KUKA KRL program: MyProgram_269().src

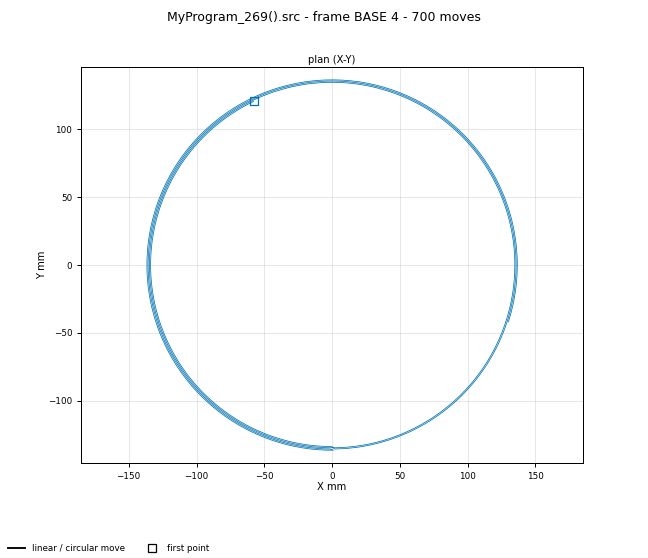
[picture p0: tool path of MyProgram_269().src in frame BASE 4, 700 of 700 moves have a stored position in this frame; points joined in program order, loops and branches not executed]
&ACCESS RVP
&REL 1
&PARAM TEMPLATE = C:\KRC\Roboter\Template\vorgabe
&PARAM EDITMASK = *
DEF MyProgram_269()
; ---- Setting reference (Base) ----
$BASE = BASE_DATA[4]

; --------------------------
; ---- Setting tool (TCP) ----
$TOOL = TOOL_DATA[3]
; --------------------------

$VEL.CP = VEL_APROX_PRINT
Startdeposition()
$VEL.CP = VEL_PRINT
LIN {X -57.9243,Y 120.6655,Z 170,A 116.7349,B 9.9654,C 0.038,E1 9.8949,E2 334.2865} C_DIS
LIN {X -61.6476,Y 118.8079,Z 170,A 118.1625,B 9.9654,C 0.0473,E1 9.8915,E2 332.903} C_DIS
LIN {X -65.3512,Y 116.8125,Z 170,A 119.9699,B 9.9654,C 0.0498,E1 9.887,E2 331.0964} C_DIS
LIN {X -69.0294,Y 114.6773,Z 170,A 121.75,B 9.9654,C 0.0533,E1 9.8828,E2 329.3227} C_DIS
LIN {X -72.8126,Y 112.3129,Z 170,A 123.7286,B 9.9654,C 0.0551,E1 9.8781,E2 327.3377} C_DIS
LIN {X -76.9825,Y 109.497,Z 170,A 126.4571,B 9.9654,C 0.0478,E1 9.8717,E2 324.5421} C_DIS
LIN {X -81.0292,Y 106.5373,Z 170,A 127.9472,B 9.9654,C 0.0641,E1 9.8685,E2 323.1329} C_DIS
LIN {X -83.788,Y 104.3816,Z 170,A 129.5953,B 9.9654,C 0.0641,E1 9.8649,E2 321.4683} C_DIS
LIN {X -86.8669,Y 101.8335,Z 170,A 131.5459,B 9.9654,C 0.0628,E1 9.8607,E2 319.4907} C_DIS
LIN {X -89.382,Y 99.6329,Z 170,A 132.7577,B 9.9653,C 0.0697,E1 9.8582,E2 318.3066} C_DIS
LIN {X -92.6442,Y 96.6073,Z 170,A 134.7532,B 9.9653,C 0.0719,E1 9.8541,E2 316.3021} C_DIS
LIN {X -95.9755,Y 93.2986,Z 170,A 136.5276,B 9.9653,C 0.0805,E1 9.8507,E2 314.5579} C_DIS
LIN {X -98.856,Y 90.2413,Z 170,A 138.5822,B 9.9653,C 0.0797,E1 9.8467,E2 312.4744} C_DIS
LIN {X -101.8694,Y 86.8246,Z 170,A 140.5352,B 9.9652,C 0.084,E1 9.8432,E2 310.5231} C_DIS
LIN {X -104.8688,Y 83.1772,Z 170,A 142.5796,B 9.9652,C 0.0882,E1 9.8396,E2 308.478} C_DIS
LIN {X -107.5965,Y 79.6178,Z 170,A 145.1791,B 9.9652,C 0.0802,E1 9.8351,E2 305.7985} C_DIS
LIN {X -110.8618,Y 75.0035,Z 170,A 147.0989,B 9.9651,C 0.0953,E1 9.8322,E2 303.9418} C_DIS
LIN {X -112.7785,Y 72.0894,Z 170,A 148.8547,B 9.9651,C 0.0943,E1 9.8295,E2 302.156} C_DIS
LIN {X -114.9795,Y 68.5242,Z 170,A 150.0203,B 9.9649,C 0.1102,E1 9.828,E2 301.0679} C_DIS
LIN {X -118.072,Y 63.0474,Z 170,A 152.9817,B 9.9649,C 0.1123,E1 9.8239,E2 298.0773} C_DIS
LIN {X -119.8941,Y 59.5049,Z 170,A 154.6712,B 9.9649,C 0.1171,E1 9.8218,E2 296.3914} C_DIS
LIN {X -121.2827,Y 56.6222,Z 170,A 155.8964,B 9.9648,C 0.1233,E1 9.8203,E2 295.1851} C_DIS
LIN {X -122.7024,Y 53.4752,Z 170,A 157.5597,B 9.9648,C 0.124,E1 9.8184,E2 293.5012} C_DIS
LIN {X -124.0518,Y 50.2648,Z 170,A 158.8105,B 9.9647,C 0.1323,E1 9.8171,E2 292.2806} C_DIS
LIN {X -126.0656,Y 44.9779,Z 170,A 161.6161,B 9.9647,C 0.1321,E1 9.8143,E2 289.4317} C_DIS
LIN {X -127.431,Y 40.9483,Z 170,A 163.3638,B 9.9646,C 0.1385,E1 9.8128,E2 287.6948} C_DIS
LIN {X -128.3886,Y 37.8391,Z 170,A 164.7682,B 9.9646,C 0.1422,E1 9.8117,E2 286.2904} C_DIS
LIN {X -129.2836,Y 34.6579,Z 170,A 166.1835,B 9.9645,C 0.1462,E1 9.8106,E2 284.8766} C_DIS
LIN {X -130.142,Y 31.2805,Z 170,A 167.7247,B 9.9645,C 0.1496,E1 9.8096,E2 283.331} C_DIS
LIN {X -130.9743,Y 27.5965,Z 170,A 169.4193,B 9.9644,C 0.1529,E1 9.8086,E2 281.6288} C_DIS
LIN {X -131.9035,Y 22.7377,Z 170,A 171.5205,B 9.9643,C 0.1592,E1 9.8075,E2 279.5318} C_DIS
LIN {X -132.4714,Y 19.1521,Z 170,A 173.0589,B 9.9642,C 0.164,E1 9.8069,E2 277.9969} C_DIS
LIN {X -132.9158,Y 15.7745,Z 170,A 174.5853,B 9.9642,C 0.167,E1 9.8063,E2 276.4638} C_DIS
LIN {X -133.3417,Y 11.6436,Z 170,A 176.4673,B 9.9641,C 0.1704,E1 9.8058,E2 274.571} C_DIS
LIN {X -133.6571,Y 7.1739,Z 170,A 178.3696,B 9.964,C 0.1762,E1 9.8055,E2 272.6725} C_DIS
LIN {X -133.8021,Y 3.5352,Z 170,A 179.8999,B 9.964,C 0.1813,E1 9.8054,E2 271.1472} C_DIS
LIN {X -133.8485,Y -0.5666,Z 170,A -178.302,B 9.9638,C 0.1857,E1 9.8054,E2 269.3458} C_DIS
LIN {X -133.7769,Y -4.4422,Z 170,A -176.5597,B 9.9638,C 0.189,E1 9.8054,E2 267.595} C_DIS
LIN {X -133.5969,Y -8.205,Z 170,A -174.9767,B 9.9637,C 0.1942,E1 9.8057,E2 266.0171} C_DIS
LIN {X -133.2712,Y -12.4241,Z 170,A -173.1406,B 9.9636,C 0.199,E1 9.8061,E2 264.1797} C_DIS
LIN {X -132.8708,Y -16.1517,Z 170,A -171.4417,B 9.9636,C 0.202,E1 9.8067,E2 262.4708} C_DIS
LIN {X -132.2959,Y -20.3285,Z 170,A -169.3217,B 9.9636,C 0.2015,E1 9.8076,E2 260.3141} C_DIS
LIN {X -131.6934,Y -23.9234,Z 170,A -167.6572,B 9.9635,C 0.2041,E1 9.8084,E2 258.6382} C_DIS
LIN {X -130.9067,Y -27.9095,Z 170,A -166.3798,B 9.9632,C 0.2174,E1 9.8091,E2 257.4187} C_DIS
LIN {X -130.1238,Y -31.3558,Z 170,A -164.4717,B 9.9632,C 0.2145,E1 9.8104,E2 255.4636} C_DIS
LIN {X -129.2659,Y -34.7243,Z 170,A -163.2928,B 9.963,C 0.2242,E1 9.8112,E2 254.3237} C_DIS
LIN {X -127.745,Y -39.9654,Z 170,A -160.7737,B 9.963,C 0.2274,E1 9.8132,E2 251.7842} C_DIS
LIN {X -126.5449,Y -43.6097,Z 170,A -159.228,B 9.9628,C 0.2336,E1 9.8146,E2 250.2517} C_DIS
LIN {X -125.4319,Y -46.7145,Z 170,A -157.8118,B 9.9628,C 0.2374,E1 9.816,E2 248.836} C_DIS
LIN {X -124.3255,Y -49.5857,Z 170,A -156.5337,B 9.9626,C 0.2416,E1 9.8173,E2 247.5636} C_DIS
LIN {X -122.9636,Y -52.8711,Z 170,A -154.9947,B 9.9626,C 0.2453,E1 9.8189,E2 246.0237} C_DIS
LIN {X -121.918,Y -55.2427,Z 170,A -153.2243,B 9.9628,C 0.2361,E1 9.8211,E2 244.1731} C_DIS
LIN {X -119.8678,Y -59.5582,Z 170,A -151.6855,B 9.9624,C 0.2507,E1 9.8229,E2 242.6978} C_DIS
LIN {X -116.8183,Y -65.3408,Z 170,A -148.7983,B 9.9623,C 0.2562,E1 9.8267,E2 239.8017} C_DIS
LIN {X -114.4677,Y -69.3759,Z 170,A -146.8451,B 9.9621,C 0.2619,E1 9.8295,E2 237.8553} C_DIS
LIN {X -112.3203,Y -72.8012,Z 170,A -144.7608,B 9.9621,C 0.2595,E1 9.8327,E2 235.7286} C_DIS
LIN {X -110.2672,Y -75.875,Z 170,A -143.4529,B 9.962,C 0.2683,E1 9.8347,E2 234.4552} C_DIS
LIN {X -107.7234,Y -79.4454,Z 170,A -141.5427,B 9.9619,C 0.272,E1 9.8379,E2 232.5419} C_DIS
LIN {X -104.8133,Y -83.2469,Z 170,A -139.4869,B 9.9617,C 0.2765,E1 9.8414,E2 230.4863} C_DIS
LIN {X -102.0403,Y -86.6235,Z 170,A -137.7705,B 9.9615,C 0.2834,E1 9.8444,E2 228.7897} C_DIS
LIN {X -99.508,Y -89.5215,Z 170,A -136.1827,B 9.9615,C 0.2881,E1 9.8473,E2 227.2099} C_DIS
LIN {X -96.878,Y -92.3609,Z 170,A -134.2445,B 9.9615,C 0.2861,E1 9.8511,E2 225.2379} C_DIS
LIN {X -94.3047,Y -94.9867,Z 170,A -132.5769,B 9.9615,C 0.2874,E1 9.8544,E2 223.5593} C_DIS
LIN {X -89.824,Y -99.2347,Z 170,A -130.0022,B 9.9612,C 0.2938,E1 9.8597,E2 220.9939} C_DIS
LIN {X -86.4166,Y -102.2162,Z 170,A -128.1722,B 9.9611,C 0.2994,E1 9.8635,E2 219.1778} C_DIS
LIN {X -82.174,Y -105.6567,Z 170,A -125.6568,B 9.9611,C 0.3,E1 9.869,E2 216.6411} C_DIS
LIN {X -79.5056,Y -107.6793,Z 170,A -123.9319,B 9.9611,C 0.2967,E1 9.873,E2 214.8805} C_DIS
LIN {X -76.5119,Y -109.8262,Z 170,A -122.6715,B 9.9609,C 0.3054,E1 9.8758,E2 213.6595} C_DIS
LIN {X -73.1187,Y -112.1142,Z 170,A -120.9687,B 9.9608,C 0.309,E1 9.8797,E2 211.9631} C_DIS
LIN {X -69.8846,Y -114.1579,Z 170,A -119.2821,B 9.9608,C 0.3104,E1 9.8837,E2 210.2706} C_DIS
LIN {X -66.9072,Y -115.9281,Z 170,A -117.781,B 9.9607,C 0.312,E1 9.8874,E2 208.7674} C_DIS
LIN {X -63.1609,Y -118.011,Z 170,A -116.0638,B 9.9605,C 0.3168,E1 9.8915,E2 207.0649} C_DIS
LIN {X -59.0597,Y -120.1137,Z 170,A -113.9364,B 9.9605,C 0.3161,E1 9.8969,E2 204.9183} C_DIS
LIN {X -55.1389,Y -121.9644,Z 170,A -112.0625,B 9.9605,C 0.3178,E1 9.9016,E2 203.0422} C_DIS
LIN {X -51.8034,Y -123.4172,Z 170,A -110.4969,B 9.9605,C 0.3192,E1 9.9057,E2 201.4755} C_DIS
LIN {X -49.0158,Y -124.5516,Z 170,A -108.7472,B 9.9607,C 0.311,E1 9.9104,E2 199.6683} C_DIS
LIN {X -44.9288,Y -126.0833,Z 170,A -107.7188,B 9.9601,C 0.3299,E1 9.9128,E2 198.744} C_DIS
LIN {X -38.134,Y -128.3023,Z 170,A -104.2346,B 9.9603,C 0.3236,E1 9.9222,E2 195.2071} C_DIS
LIN {X -34.1836,Y -129.4101,Z 170,A -102.4939,B 9.9603,C 0.325,E1 9.9269,E2 193.468} C_DIS
LIN {X -30.0866,Y -130.4234,Z 170,A -100.6752,B 9.9603,C 0.3258,E1 9.9318,E2 191.6474} C_DIS
LIN {X -26.4187,Y -131.2156,Z 170,A -99.0363,B 9.9603,C 0.3258,E1 9.9363,E2 190.004} C_DIS
LIN {X -22.1834,Y -131.9975,Z 170,A -97.2401,B 9.9603,C 0.3276,E1 9.9412,E2 188.2132} C_DIS
LIN {X -18.358,Y -132.5849,Z 170,A -95.4984,B 9.9603,C 0.3263,E1 9.9461,E2 186.4604} C_DIS
LIN {X -14.1661,Y -133.0969,Z 170,A -93.7824,B 9.9602,C 0.3286,E1 9.9508,E2 184.7551} C_DIS
LIN {X -9.9819,Y -133.4761,Z 170,A -92.0352,B 9.9602,C 0.3299,E1 9.9557,E2 183.0137} C_DIS
LIN {X -5.8315,Y -133.723,Z 170,A -89.4693,B 9.9607,C 0.313,E1 9.9631,E2 180.3486} C_DIS
LIN {X -0.1381,Y -133.85,Z 170,A -87.6713,B 9.9602,C 0.3266,E1 9.9679,E2 178.6297} C_DIS
LIN {X -0.1381,Y -133.85,Z 170,A -87.6713,B 9.9602,C 0.3266,E1 9.9679,E2 178.6297} C_DIS
Enddeposition()
LIN {X 0.9771,Y -134.7546,Z 170,A -87.4135,B 9.7192,C 0.3449,E1 9.728,E2 178.5039} C_DIS
Startdeposition()
$VEL.CP = VEL_PRINT
LIN {X -4.4951,Y -134.6861,Z 170,A -90.2098,B 9.7189,C 0.3551,E1 9.72,E2 181.3599} C_DIS
LIN {X -8.9106,Y -134.467,Z 170,A -92.1285,B 9.7189,C 0.3558,E1 9.7146,E2 183.2843} C_DIS
LIN {X -12.8261,Y -134.1486,Z 170,A -93.73,B 9.7189,C 0.3541,E1 9.7102,E2 184.8779} C_DIS
LIN {X -16.5143,Y -133.7458,Z 170,A -95.3898,B 9.7189,C 0.3555,E1 9.7056,E2 186.5485} C_DIS
LIN {X -20.4759,Y -133.1957,Z 170,A -97.0229,B 9.7189,C 0.3536,E1 9.7011,E2 188.1738} C_DIS
LIN {X -24.06,Y -132.5954,Z 170,A -98.6614,B 9.7189,C 0.3549,E1 9.6965,E2 189.8243} C_DIS
LIN {X -28.2967,Y -131.7559,Z 170,A -100.3974,B 9.7189,C 0.352,E1 9.6918,E2 191.5483} C_DIS
LIN {X -31.5958,Y -131.0038,Z 170,A -101.8668,B 9.7189,C 0.3519,E1 9.6878,E2 193.022} C_DIS
LIN {X -35.6382,Y -129.9641,Z 170,A -103.6858,B 9.7189,C 0.3517,E1 9.6829,E2 194.8468} C_DIS
LIN {X -38.8872,Y -129.0287,Z 170,A -105.798,B 9.7185,C 0.3641,E1 9.677,E2 197.0422} C_DIS
LIN {X -44.1155,Y -127.3346,Z 170,A -107.404,B 9.7191,C 0.3477,E1 9.673,E2 198.5587} C_DIS
LIN {X -47.4018,Y -126.1481,Z 170,A -109.1766,B 9.719,C 0.352,E1 9.6683,E2 200.3669} C_DIS
LIN {X -51.7755,Y -124.4169,Z 170,A -110.9075,B 9.7192,C 0.3448,E1 9.6639,E2 202.0649} C_DIS
LIN {X -54.7429,Y -123.1404,Z 170,A -112.3141,B 9.7192,C 0.344,E1 9.6603,E2 203.4756} C_DIS
LIN {X -57.5955,Y -121.833,Z 170,A -113.5226,B 9.7194,C 0.34,E1 9.6572,E2 204.6686} C_DIS
LIN {X -62.2414,Y -119.5259,Z 170,A -115.9406,B 9.7194,C 0.3415,E1 9.6512,E2 207.1128} C_DIS
LIN {X -66.0211,Y -117.4819,Z 170,A -117.7294,B 9.7194,C 0.3384,E1 9.6468,E2 208.8969} C_DIS
LIN {X -69.3149,Y -115.5697,Z 170,A -119.2947,B 9.7196,C 0.3351,E1 9.643,E2 210.4555} C_DIS
LIN {X -72.4733,Y -113.6153,Z 170,A -121.0175,B 9.7196,C 0.3356,E1 9.6389,E2 212.1957} C_DIS
LIN {X -76.11,Y -111.2118,Z 170,A -122.7076,B 9.7198,C 0.3297,E1 9.635,E2 213.8654} C_DIS
LIN {X -81.907,Y -107.0141,Z 170,A -125.7083,B 9.7199,C 0.3239,E1 9.6283,E2 216.8604} C_DIS
LIN {X -86.3855,Y -103.4331,Z 170,A -128.446,B 9.7199,C 0.3253,E1 9.6223,E2 219.6344} C_DIS
LIN {X -89.9009,Y -100.3922,Z 170,A -130.333,B 9.7201,C 0.32,E1 9.6183,E2 221.5099} C_DIS
LIN {X -93.4041,Y -97.1422,Z 170,A -132.2223,B 9.7203,C 0.3135,E1 9.6145,E2 223.3812} C_DIS
LIN {X -95.7296,Y -94.8507,Z 170,A -133.8096,B 9.7203,C 0.3145,E1 9.6113,E2 224.9924} C_DIS
LIN {X -98.151,Y -92.3427,Z 170,A -135.5462,B 9.7203,C 0.3161,E1 9.6079,E2 226.7595} C_DIS
LIN {X -102.1954,Y -87.8457,Z 170,A -137.9522,B 9.7205,C 0.3077,E1 9.6035,E2 229.1443} C_DIS
LIN {X -105.0155,Y -84.4545,Z 170,A -139.8374,B 9.7205,C 0.3037,E1 9.6002,E2 231.0298} C_DIS
LIN {X -107.7253,Y -80.9697,Z 170,A -141.7675,B 9.7207,C 0.3005,E1 9.5969,E2 232.9655} C_DIS
LIN {X -110.2855,Y -77.4465,Z 170,A -143.6834,B 9.7207,C 0.2974,E1 9.5938,E2 234.8883} C_DIS
LIN {X -113.403,Y -72.8049,Z 170,A -146.0574,B 9.721,C 0.2917,E1 9.5901,E2 237.2606} C_DIS
LIN {X -115.8267,Y -68.8837,Z 170,A -148.0148,B 9.721,C 0.2869,E1 9.5873,E2 239.2166} C_DIS
LIN {X -117.92,Y -65.2354,Z 170,A -150.3141,B 9.721,C 0.2915,E1 9.5841,E2 241.5766} C_DIS
LIN {X -120.0516,Y -61.2196,Z 170,A -151.6792,B 9.7214,C 0.2765,E1 9.5824,E2 242.8716} C_DIS
LIN {X -122.7954,Y -55.5141,Z 170,A -154.5067,B 9.7215,C 0.2719,E1 9.579,E2 245.7139} C_DIS
LIN {X -124.2821,Y -52.0984,Z 170,A -155.9847,B 9.7217,C 0.2659,E1 9.5774,E2 247.1778} C_DIS
LIN {X -125.4871,Y -49.1259,Z 170,A -157.4166,B 9.7217,C 0.2634,E1 9.5759,E2 248.6171} C_DIS
LIN {X -126.5852,Y -46.2249,Z 170,A -158.8446,B 9.7217,C 0.2618,E1 9.5745,E2 250.0574} C_DIS
LIN {X -127.7861,Y -42.7907,Z 170,A -160.2742,B 9.722,C 0.2555,E1 9.5733,E2 251.4716} C_DIS
LIN {X -130,Y -35.5095,Z 170,A -164.2806,B 9.7218,C 0.26,E1 9.5701,E2 255.5684} C_DIS
LIN {X -131.2504,Y -30.5605,Z 170,A -165.8723,B 9.7223,C 0.2439,E1 9.5691,E2 257.0887} C_DIS
LIN {X -132.0168,Y -27.0538,Z 170,A -167.3025,B 9.7224,C 0.2379,E1 9.5683,E2 258.5059} C_DIS
LIN {X -133.1512,Y -20.7629,Z 170,A -170.1331,B 9.7225,C 0.2321,E1 9.5669,E2 261.3479} C_DIS
LIN {X -133.6462,Y -17.2942,Z 170,A -171.6623,B 9.7226,C 0.2285,E1 9.5663,E2 262.8805} C_DIS
LIN {X -134.1146,Y -13.1804,Z 170,A -173.4507,B 9.7227,C 0.2239,E1 9.5658,E2 264.6707} C_DIS
LIN {X -134.4217,Y -9.5513,Z 170,A -175.0694,B 9.7228,C 0.2206,E1 9.5654,E2 266.2964} C_DIS
LIN {X -134.6475,Y -5.5229,Z 170,A -176.7595,B 9.7229,C 0.2152,E1 9.5652,E2 267.9819} C_DIS
LIN {X -134.7544,Y -1.4756,Z 170,A -178.5057,B 9.723,C 0.2106,E1 9.5651,E2 269.7295} C_DIS
LIN {X -134.7396,Y 2.379,Z 170,A 179.7909,B 9.7231,C 0.2069,E1 9.5651,E2 271.439} C_DIS
LIN {X -134.6023,Y 6.5307,Z 170,A 178.0437,B 9.7232,C 0.2015,E1 9.5653,E2 273.1822} C_DIS
LIN {X -134.3987,Y 9.8665,Z 170,A 176.5566,B 9.7232,C 0.1985,E1 9.5656,E2 274.6759} C_DIS
LIN {X -134.0277,Y 14.0378,Z 170,A 174.7855,B 9.7234,C 0.1931,E1 9.5661,E2 276.4441} C_DIS
LIN {X -133.626,Y 17.4478,Z 170,A 173.3066,B 9.7234,C 0.1892,E1 9.5666,E2 277.9238} C_DIS
LIN {X -133.0718,Y 21.2758,Z 170,A 171.3681,B 9.7234,C 0.1896,E1 9.5674,E2 279.8959} C_DIS
LIN {X -132.2236,Y 26.0331,Z 170,A 169.4074,B 9.7236,C 0.182,E1 9.5684,E2 281.8433} C_DIS
LIN {X -131.4843,Y 29.5367,Z 170,A 168.0015,B 9.7237,C 0.1757,E1 9.5693,E2 283.2336} C_DIS
LIN {X -130.6161,Y 33.1621,Z 170,A 166.3806,B 9.7237,C 0.1718,E1 9.5704,E2 284.857} C_DIS
LIN {X -129.5444,Y 37.1365,Z 170,A 164.5101,B 9.7238,C 0.1689,E1 9.5718,E2 286.7402} C_DIS
LIN {X -128.4954,Y 40.6125,Z 170,A 163.0045,B 9.7239,C 0.1639,E1 9.573,E2 288.2395} C_DIS
LIN {X -127.4386,Y 43.8154,Z 170,A 161.1752,B 9.7239,C 0.1668,E1 9.5747,E2 290.1145} C_DIS
LIN {X -126.1073,Y 47.5108,Z 170,A 159.8117,B 9.724,C 0.1569,E1 9.576,E2 291.4397} C_DIS
LIN {X -124.4401,Y 51.72,Z 170,A 158.1735,B 9.7242,C 0.1467,E1 9.5777,E2 293.0415} C_DIS
LIN {X -123.2292,Y 54.5443,Z 170,A 156.5305,B 9.7242,C 0.149,E1 9.5795,E2 294.7234} C_DIS
LIN {X -121.6379,Y 58.0039,Z 170,A 155.0064,B 9.7242,C 0.143,E1 9.5813,E2 296.2345} C_DIS
LIN {X -120.0489,Y 61.225,Z 170,A 153.4683,B 9.7243,C 0.1392,E1 9.5832,E2 297.7722} C_DIS
LIN {X -117.0904,Y 66.7129,Z 170,A 150.7299,B 9.7243,C 0.1339,E1 9.5869,E2 300.5184} C_DIS
LIN {X -115.0176,Y 70.2268,Z 170,A 148.9131,B 9.7244,C 0.131,E1 9.5895,E2 302.3432} C_DIS
LIN {X -112.6799,Y 73.9193,Z 170,A 147.1169,B 9.7244,C 0.1253,E1 9.5922,E2 304.13} C_DIS
LIN {X -108.6836,Y 79.6786,Z 170,A 143.9959,B 9.7245,C 0.1206,E1 9.5973,E2 307.2646} C_DIS
LIN {X -106.0447,Y 83.1583,Z 170,A 142.1258,B 9.7245,C 0.1165,E1 9.6005,E2 309.1344} C_DIS
LIN {X -103.1639,Y 86.7063,Z 170,A 140.1101,B 9.7246,C 0.1134,E1 9.6041,E2 311.1568} C_DIS
LIN {X -100.0761,Y 90.2536,Z 170,A 138.0969,B 9.7246,C 0.1092,E1 9.6078,E2 313.1696} C_DIS
LIN {X -96.8003,Y 93.7575,Z 170,A 136.0795,B 9.7247,C 0.1044,E1 9.6117,E2 315.1822} C_DIS
LIN {X -94.1463,Y 96.4227,Z 170,A 134.4473,B 9.7247,C 0.1017,E1 9.6149,E2 316.8168} C_DIS
LIN {X -90.878,Y 99.5095,Z 170,A 132.4755,B 9.7247,C 0.0989,E1 9.6189,E2 318.7938} C_DIS
LIN {X -87.125,Y 102.8107,Z 170,A 130.3875,B 9.7248,C 0.0941,E1 9.6233,E2 320.8754} C_DIS
LIN {X -83.7824,Y 105.5524,Z 170,A 128.7514,B 9.7249,C 0.087,E1 9.6268,E2 322.4857} C_DIS
LIN {X -78.8326,Y 109.2991,Z 170,A 125.9998,B 9.7249,C 0.0844,E1 9.633,E2 325.2482} C_DIS
LIN {X -75.7767,Y 111.4394,Z 170,A 124.2328,B 9.7249,C 0.085,E1 9.6371,E2 327.0353} C_DIS
LIN {X -72.2613,Y 113.7507,Z 170,A 122.4507,B 9.7249,C 0.082,E1 9.6413,E2 328.815} C_DIS
LIN {X -69.1255,Y 115.6826,Z 170,A 120.8478,B 9.7249,C 0.0803,E1 9.6451,E2 330.4209} C_DIS
LIN {X -65.1242,Y 117.9815,Z 170,A 118.9022,B 9.7249,C 0.0771,E1 9.6498,E2 332.3628} C_DIS
LIN {X -60.4576,Y 120.4376,Z 170,A 116.4291,B 9.7249,C 0.0784,E1 9.6561,E2 334.8614} C_DIS
LIN {X -57.4113,Y 121.9211,Z 170,A 115.2085,B 9.725,C 0.0724,E1 9.6591,E2 336.0547} C_DIS
LIN {X -53.931,Y 123.4987,Z 170,A 113.6182,B 9.725,C 0.0698,E1 9.6631,E2 337.6396} C_DIS
LIN {X -50.2829,Y 125.0276,Z 170,A 110.7916,B 9.7249,C 0.0894,E1 9.6708,E2 340.5996} C_DIS
LIN {X -42.9936,Y 127.7185,Z 170,A 108.5673,B 9.7251,C 0.0658,E1 9.6763,E2 342.6946} C_DIS
LIN {X -34.2182,Y 130.3445,Z 170,A 104.6068,B 9.7251,C 0.0638,E1 9.687,E2 346.6603} C_DIS
LIN {X -30.2257,Y 131.3269,Z 170,A 102.9816,B 9.7251,C 0.0601,E1 9.6913,E2 348.2697} C_DIS
LIN {X -26.7634,Y 132.0759,Z 170,A 101.3934,B 9.7251,C 0.0608,E1 9.6957,E2 349.8667} C_DIS
LIN {X -22.4296,Y 132.8808,Z 170,A 99.5235,B 9.7251,C 0.0597,E1 9.7008,E2 351.7349} C_DIS
LIN {X -18.9606,Y 133.4198,Z 170,A 98.0625,B 9.7251,C 0.0584,E1 9.7048,E2 353.1913} C_DIS
LIN {X -14.9666,Y 133.9278,Z 170,A 96.2689,B 9.7251,C 0.0593,E1 9.7098,E2 354.9937} C_DIS
LIN {X -11.5126,Y 134.2678,Z 170,A 94.9181,B 9.7251,C 0.0564,E1 9.7135,E2 356.3288} C_DIS
LIN {X -8.2991,Y 134.5046,Z 170,A 93.497,B 9.7251,C 0.0571,E1 9.7175,E2 357.7553} C_DIS
LIN {X -4.3993,Y 134.6902,Z 170,A 91.7459,B 9.7251,C 0.0587,E1 9.7224,E2 359.5164} C_DIS
LIN {X -0.5579,Y 134.7595,Z 170,A 90.2192,B 9.7251,C 0.0564,E1 9.7267,E2 361.0297} C_DIS
LIN {X 3.0963,Y 134.7265,Z 170,A 88.5578,B 9.7251,C 0.0586,E1 9.7313,E2 362.7032} C_DIS
LIN {X 7.1572,Y 134.5708,Z 170,A 86.802,B 9.7251,C 0.0594,E1 9.7362,E2 364.4616} C_DIS
LIN {X 11.2305,Y 134.2917,Z 170,A 85.1526,B 9.7251,C 0.0579,E1 9.7408,E2 366.1} C_DIS
LIN {X 15.3754,Y 133.8816,Z 170,A 83.3198,B 9.7251,C 0.0597,E1 9.7459,E2 367.9397} C_DIS
LIN {X 19.2035,Y 133.3851,Z 170,A 81.8206,B 9.7251,C 0.0574,E1 9.75,E2 369.4213} C_DIS
LIN {X 22.3521,Y 132.8937,Z 170,A 80.3941,B 9.7251,C 0.0594,E1 9.754,E2 370.8559} C_DIS
LIN {X 26.5055,Y 132.1284,Z 170,A 78.6392,B 9.7251,C 0.0595,E1 9.7588,E2 372.6055} C_DIS
LIN {X 29.9893,Y 131.3809,Z 170,A 77.108,B 9.7251,C 0.0608,E1 9.7629,E2 374.1382} C_DIS
LIN {X 33.612,Y 130.5019,Z 170,A 75.477,B 9.7251,C 0.0628,E1 9.7674,E2 375.7745} C_DIS
LIN {X 41.0357,Y 128.3602,Z 170,A 72.2905,B 9.7251,C 0.0633,E1 9.7759,E2 378.9487} C_DIS
LIN {X 44.6111,Y 127.1627,Z 170,A 70.4353,B 9.7251,C 0.0702,E1 9.7809,E2 380.8338} C_DIS
LIN {X 48.972,Y 125.5469,Z 170,A 68.7154,B 9.7251,C 0.0667,E1 9.7853,E2 382.5228} C_DIS
LIN {X 52.7591,Y 124.0054,Z 170,A 66.8706,B 9.7251,C 0.0708,E1 9.7901,E2 384.3802} C_DIS
LIN {X 56.2147,Y 122.4757,Z 170,A 65.4282,B 9.7251,C 0.0692,E1 9.7937,E2 385.8029} C_DIS
LIN {X 59.2847,Y 121.0194,Z 170,A 63.9188,B 9.7251,C 0.0723,E1 9.7975,E2 387.3201} C_DIS
LIN {X 62.462,Y 119.4101,Z 170,A 62.4453,B 9.7251,C 0.0734,E1 9.8011,E2 388.7887} C_DIS
LIN {X 66.2679,Y 117.3432,Z 170,A 60.6612,B 9.7251,C 0.0747,E1 9.8055,E2 390.5661} C_DIS
LIN {X 68.8541,Y 115.8444,Z 170,A 59.2954,B 9.725,C 0.0786,E1 9.8088,E2 391.9434} C_DIS
LIN {X 72.4733,Y 113.6153,Z 170,A 57.494,B 9.725,C 0.0812,E1 9.8131,E2 393.7443} C_DIS
LIN {X 78.1668,Y 109.7761,Z 170,A 54.5608,B 9.725,C 0.0863,E1 9.8198,E2 396.6797} C_DIS
LIN {X 81.617,Y 107.2359,Z 170,A 52.6745,B 9.7249,C 0.0908,E1 9.8241,E2 398.5741} C_DIS
LIN {X 85.5189,Y 104.1508,Z 170,A 50.6756,B 9.7249,C 0.092,E1 9.8284,E2 400.5596} C_DIS
LIN {X 88.8945,Y 101.2851,Z 170,A 48.7663,B 9.7249,C 0.0962,E1 9.8324,E2 402.4727} C_DIS
LIN {X 92.3929,Y 98.1037,Z 170,A 46.8346,B 9.7248,C 0.0983,E1 9.8364,E2 404.3955} C_DIS
LIN {X 95.6294,Y 94.9515,Z 170,A 44.8522,B 9.7248,C 0.1036,E1 9.8403,E2 406.386} C_DIS
LIN {X 98.9728,Y 91.4619,Z 170,A 42.8564,B 9.7248,C 0.1065,E1 9.8441,E2 408.3755} C_DIS
LIN {X 101.8721,Y 88.2212,Z 170,A 41.0725,B 9.7247,C 0.109,E1 9.8474,E2 410.1523} C_DIS
LIN {X 103.9422,Y 85.772,Z 170,A 39.1696,B 9.7245,C 0.1243,E1 9.8509,E2 412.1207} C_DIS
LIN {X 107.142,Y 81.7397,Z 170,A 37.5657,B 9.7246,C 0.116,E1 9.8535,E2 413.6554} C_DIS
LIN {X 109.6293,Y 78.372,Z 170,A 35.6235,B 9.7246,C 0.1239,E1 9.8567,E2 415.6181} C_DIS
LIN {X 112.7671,Y 73.7868,Z 170,A 33.4779,B 9.7246,C 0.1245,E1 9.86,E2 417.7388} C_DIS
LIN {X 115.0055,Y 70.2465,Z 170,A 31.7538,B 9.7245,C 0.1276,E1 9.8626,E2 419.4571} C_DIS
LIN {X 117.1796,Y 66.556,Z 170,A 29.6398,B 9.7243,C 0.1389,E1 9.8656,E2 421.6076} C_DIS
LIN {X 118.9531,Y 63.3323,Z 170,A 28.3353,B 9.7243,C 0.1369,E1 9.8672,E2 422.8817} C_DIS
LIN {X 120.6368,Y 60.0603,Z 170,A 26.8561,B 9.7243,C 0.1389,E1 9.8691,E2 424.3515} C_DIS
LIN {X 122.203,Y 56.8043,Z 170,A 25.3984,B 9.7243,C 0.1411,E1 9.8708,E2 425.8007} C_DIS
LIN {X 123.6433,Y 53.5966,Z 170,A 23.9427,B 9.7243,C 0.1441,E1 9.8725,E2 427.2526} C_DIS
LIN {X 125.2323,Y 49.7751,Z 170,A 21.6294,B 9.724,C 0.1618,E1 9.8749,E2 429.6344} C_DIS
LIN {X 126.8753,Y 45.4204,Z 170,A 20.2047,B 9.724,C 0.1542,E1 9.8762,E2 430.9934} C_DIS
LIN {X 128.2042,Y 41.5241,Z 170,A 17.8097,B 9.7237,C 0.1741,E1 9.8784,E2 433.4678} C_DIS
LIN {X 129.7748,Y 36.3151,Z 170,A 16.2523,B 9.7239,C 0.1628,E1 9.8795,E2 434.9355} C_DIS
LIN {X 130.6299,Y 33.1077,Z 170,A 14.841,B 9.7239,C 0.1668,E1 9.8805,E2 436.348} C_DIS
LIN {X 131.5367,Y 29.3071,Z 170,A 13.1174,B 9.7238,C 0.173,E1 9.8816,E2 438.0807} C_DIS
LIN {X 132.3205,Y 25.5275,Z 170,A 11.6108,B 9.7238,C 0.1745,E1 9.8824,E2 439.5722} C_DIS
LIN {X 132.93,Y 22.1345,Z 170,A 10.1412,B 9.7237,C 0.1787,E1 9.8831,E2 441.0435} C_DIS
LIN {X 133.5316,Y 18.1688,Z 170,A 8.5033,B 9.7237,C 0.1821,E1 9.8838,E2 442.6748} C_DIS
LIN {X 133.9501,Y 14.7589,Z 170,A 7.0038,B 9.7235,C 0.1872,E1 9.8843,E2 444.1803} C_DIS
LIN {X 134.298,Y 11.1553,Z 170,A 5.4631,B 9.7235,C 0.1917,E1 9.8846,E2 445.7226} C_DIS
LIN {X 134.5748,Y 7.0779,Z 170,A 3.7664,B 9.7233,C 0.1958,E1 9.8849,E2 447.4159} C_DIS
LIN {X 134.7244,Y 3.1698,Z 170,A 2.0941,B 9.7233,C 0.2008,E1 9.8851,E2 449.091} C_DIS
LIN {X 134.761,Y -0.4414,Z 170,A 0.5387,B 9.7231,C 0.2058,E1 9.8851,E2 450.6503} C_DIS
LIN {X 134.6752,Y -4.8135,Z 170,A -1.0247,B 9.7231,C 0.2042,E1 9.885,E2 452.1792} C_DIS
LIN {X 134.5482,Y -7.5925,Z 170,A -2.4378,B 9.723,C 0.2131,E1 9.8848,E2 453.6218} C_DIS
LIN {X 134.2781,Y -11.3915,Z 170,A -3.9793,B 9.723,C 0.216,E1 9.8844,E2 455.1553} C_DIS
LIN {X 133.8576,Y -15.5767,Z 170,A -5.759,B 9.7228,C 0.221,E1 9.8839,E2 456.9358} C_DIS
LIN {X 133.3506,Y -19.4451,Z 170,A -7.4625,B 9.7227,C 0.2269,E1 9.8832,E2 458.6465} C_DIS
LIN {X 132.6563,Y -23.7196,Z 170,A -9.1637,B 9.7227,C 0.2288,E1 9.8825,E2 460.3324} C_DIS
LIN {X 131.9196,Y -27.5316,Z 170,A -10.9147,B 9.7225,C 0.236,E1 9.8815,E2 462.0975} C_DIS
LIN {X 130.9961,Y -31.6279,Z 170,A -13.3368,B 9.7219,C 0.2561,E1 9.8799,E2 464.5991} C_DIS
LIN {X 129.447,Y -37.4691,Z 170,A -15.0104,B 9.7223,C 0.2422,E1 9.8787,E2 466.166} C_DIS
LIN {X 128.4866,Y -40.6399,Z 170,A -16.4344,B 9.7222,C 0.2466,E1 9.8775,E2 467.5934} C_DIS
LIN {X 127.501,Y -43.6354,Z 170,A -17.9913,B 9.722,C 0.2555,E1 9.8761,E2 469.1784} C_DIS
LIN {X 125.7708,Y -48.3961,Z 170,A -19.8937,B 9.722,C 0.2555,E1 9.8742,E2 471.0521} C_DIS
LIN {X 124.4038,Y -51.807,Z 170,A -21.4219,B 9.7219,C 0.2589,E1 9.8726,E2 472.5777} C_DIS
LIN {X 123.2292,Y -54.5443,Z 170,A -23.6416,B 9.7212,C 0.2848,E1 9.87,E2 474.9156} C_DIS
LIN {X 120.3106,Y -60.7109,Z 170,A -25.6096,B 9.7216,C 0.2706,E1 9.8677,E2 476.7727} C_DIS
LIN {X 118.4923,Y -64.1911,Z 170,A -27.9211,B 9.721,C 0.2901,E1 9.8645,E2 479.1648} C_DIS
LIN {X 115.7314,Y -69.0437,Z 170,A -29.5903,B 9.7213,C 0.2797,E1 9.8623,E2 480.7501} C_DIS
LIN {X 113.5225,Y -72.6183,Z 170,A -31.343,B 9.7213,C 0.2834,E1 9.8597,E2 482.5005} C_DIS
LIN {X 111.2686,Y -76.0273,Z 170,A -33.4986,B 9.7208,C 0.2975,E1 9.8562,E2 484.7095} C_DIS
LIN {X 108.7802,Y -79.547,Z 170,A -34.7233,B 9.7211,C 0.2877,E1 9.8543,E2 485.8612} C_DIS
LIN {X 106.0626,Y -83.1355,Z 170,A -36.8154,B 9.7208,C 0.2964,E1 9.8507,E2 487.9775} C_DIS
LIN {X 103.8118,Y -85.9295,Z 170,A -38.5222,B 9.7206,C 0.3042,E1 9.8477,E2 489.7082} C_DIS
LIN {X 101.6533,Y -88.4726,Z 170,A -39.7263,B 9.7206,C 0.3025,E1 9.8455,E2 490.8875} C_DIS
LIN {X 98.556,Y -91.9103,Z 170,A -41.6939,B 9.7205,C 0.3069,E1 9.8418,E2 492.8571} C_DIS
LIN {X 95.2915,Y -95.2915,Z 170,A -43.3853,B 9.7205,C 0.3041,E1 9.8386,E2 494.5125} C_DIS
LIN {X 92.6636,Y -97.8483,Z 170,A -45.1736,B 9.7203,C 0.3127,E1 9.8349,E2 496.3309} C_DIS
LIN {X 89.3643,Y -100.8702,Z 170,A -47.056,B 9.7203,C 0.3161,E1 9.831,E2 498.2127} C_DIS
LIN {X 86.0826,Y -103.685,Z 170,A -48.8581,B 9.7201,C 0.3189,E1 9.8271,E2 500.0122} C_DIS
LIN {X 80.8541,Y -107.8125,Z 170,A -51.7108,B 9.7199,C 0.3247,E1 9.8209,E2 502.8701} C_DIS
LIN {X 75.7964,Y -111.4261,Z 170,A -54.3343,B 9.7198,C 0.3289,E1 9.8149,E2 505.4937} C_DIS
LIN {X 72.0127,Y -113.9077,Z 170,A -56.1984,B 9.7198,C 0.3308,E1 9.8105,E2 507.3522} C_DIS
LIN {X 65.3454,Y -117.8591,Z 170,A -59.3871,B 9.7196,C 0.3336,E1 9.8028,E2 510.5307} C_DIS
LIN {X 61.6811,Y -119.8167,Z 170,A -61.0631,B 9.7196,C 0.3341,E1 9.7987,E2 512.197} C_DIS
LIN {X 58.9593,Y -121.1799,Z 170,A -62.7075,B 9.7193,C 0.3438,E1 9.7945,E2 513.886} C_DIS
LIN {X 53.8854,Y -123.5184,Z 170,A -64.7938,B 9.7193,C 0.3404,E1 9.7892,E2 515.9384} C_DIS
LIN {X 50.4666,Y -124.9535,Z 170,A -66.6925,B 9.7191,C 0.3495,E1 9.7842,E2 517.8782} C_DIS
LIN {X 47.1541,Y -126.2409,Z 170,A -67.9031,B 9.7192,C 0.3446,E1 9.7812,E2 519.0529} C_DIS
LIN {X 43.5044,Y -127.5464,Z 170,A -69.4883,B 9.7192,C 0.345,E1 9.777,E2 520.6316} C_DIS
LIN {X 39.7151,Y -128.7753,Z 170,A -71.1167,B 9.7192,C 0.3453,E1 9.7727,E2 522.2531} C_DIS
LIN {X 36.1,Y -129.835,Z 170,A -72.8885,B 9.719,C 0.3504,E1 9.7679,E2 524.0471} C_DIS
LIN {X 31.7751,Y -130.9606,Z 170,A -74.6639,B 9.719,C 0.3493,E1 9.7631,E2 525.8084} C_DIS
LIN {X 28.5512,Y -131.701,Z 170,A -76.0798,B 9.719,C 0.3506,E1 9.7592,E2 527.2265} C_DIS
LIN {X 24.47,Y -132.522,Z 170,A -77.9132,B 9.719,C 0.3532,E1 9.7542,E2 529.069} C_DIS
LIN {X 20.6072,Y -133.1753,Z 170,A -79.4899,B 9.719,C 0.3522,E1 9.7499,E2 530.6356} C_DIS
LIN {X 16.8127,Y -133.7093,Z 170,A -81.2382,B 9.7188,C 0.3556,E1 9.745,E2 532.3998} C_DIS
LIN {X 12.9135,Y -134.1402,Z 170,A -82.7788,B 9.7189,C 0.3536,E1 9.7407,E2 533.9255} C_DIS
LIN {X 8.8712,Y -134.4694,Z 170,A -85.0901,B 9.7184,C 0.3666,E1 9.7341,E2 536.3102} C_DIS
LIN {X 4.0559,Y -134.6998,Z 170,A -86.5869,B 9.7189,C 0.3554,E1 9.7301,E2 537.7399} C_DIS
LIN {X 0.9771,Y -134.7546,Z 170,A -87.4108,B 9.7192,C 0.3454,E1 9.728,E2 538.5038} C_DIS
Enddeposition()
LIN {X 0.9771,Y -134.7546,Z 170,A -87.4108,B 9.7192,C 0.3454,E1 9.728,E2 538.5038} C_DIS
Startdeposition()
$VEL.CP = VEL_PRINT
LIN {X 1.5938,Y -135.6645,Z 170,A -86.9648,B 9.6522,C 0.3492,E1 9.6623,E2 538.0882} C_DIS
LIN {X 8.6475,Y -135.3967,Z 170,A -84.0297,B 9.6522,C 0.3495,E1 9.6705,E2 535.1576} C_DIS
LIN {X 12.1264,Y -135.131,Z 170,A -82.4742,B 9.6522,C 0.3472,E1 9.6749,E2 533.5909} C_DIS
LIN {X 15.7984,Y -134.7494,Z 170,A -80.879,B 9.6524,C 0.3457,E1 9.6793,E2 531.9903} C_DIS
LIN {X 18.8367,Y -134.3585,Z 170,A -79.7101,B 9.6523,C 0.3477,E1 9.6825,E2 530.8363} C_DIS
LIN {X 21.4312,Y -133.9704,Z 170,A -78.3746,B 9.6525,C 0.3422,E1 9.6863,E2 529.4714} C_DIS
LIN {X 25.1418,Y -133.3225,Z 170,A -76.9844,B 9.6524,C 0.3455,E1 9.69,E2 528.1055} C_DIS
LIN {X 28.3993,Y -132.6665,Z 170,A -75.5194,B 9.6524,C 0.3432,E1 9.694,E2 526.6318} C_DIS
LIN {X 31.6943,Y -131.918,Z 170,A -74.1043,B 9.6524,C 0.3423,E1 9.6979,E2 525.2172} C_DIS
LIN {X 34.7785,Y -131.1387,Z 170,A -72.6925,B 9.6526,C 0.3396,E1 9.7017,E2 523.7958} C_DIS
LIN {X 38.9856,Y -129.9521,Z 170,A -70.9334,B 9.6526,C 0.3399,E1 9.7064,E2 522.0464} C_DIS
LIN {X 41.7717,Y -129.0822,Z 170,A -69.5361,B 9.6527,C 0.3349,E1 9.7102,E2 520.6273} C_DIS
LIN {X 45.3709,Y -127.8624,Z 170,A -68.1567,B 9.6527,C 0.3383,E1 9.7138,E2 519.2753} C_DIS
LIN {X 48.6481,Y -126.651,Z 170,A -66.5648,B 9.6527,C 0.334,E1 9.718,E2 517.6675} C_DIS
LIN {X 52.1635,Y -125.243,Z 170,A -65.0358,B 9.6527,C 0.3336,E1 9.7219,E2 516.1461} C_DIS
LIN {X 55.1155,Y -123.9725,Z 170,A -63.5972,B 9.6529,C 0.33,E1 9.7256,E2 514.696} C_DIS
LIN {X 59.1306,Y -122.1101,Z 170,A -61.8464,B 9.6529,C 0.3302,E1 9.73,E2 512.9587} C_DIS
LIN {X 62.5616,Y -120.3876,Z 170,A -60.3278,B 9.6529,C 0.3302,E1 9.7337,E2 511.4517} C_DIS
LIN {X 64.9881,Y -119.0962,Z 170,A -58.974,B 9.6531,C 0.3241,E1 9.7371,E2 510.0724} C_DIS
LIN {X 67.6578,Y -117.6006,Z 170,A -57.5222,B 9.6533,C 0.3184,E1 9.7407,E2 508.5993} C_DIS
LIN {X 71.9823,Y -115.0044,Z 170,A -55.6117,B 9.6533,C 0.32,E1 9.7452,E2 506.7147} C_DIS
LIN {X 75.6657,Y -112.6153,Z 170,A -53.9927,B 9.6532,C 0.3222,E1 9.7489,E2 505.1238} C_DIS
LIN {X 78.333,Y -110.776,Z 170,A -52.485,B 9.6533,C 0.3166,E1 9.7524,E2 503.5971} C_DIS
LIN {X 81.4942,Y -108.4718,Z 170,A -50.8499,B 9.6534,C 0.314,E1 9.7561,E2 501.9626} C_DIS
LIN {X 84.8952,Y -105.8313,Z 170,A -48.9243,B 9.6536,C 0.3081,E1 9.7603,E2 500.0217} C_DIS
LIN {X 88.3934,Y -102.9271,Z 170,A -47.0872,B 9.6536,C 0.3062,E1 9.7642,E2 498.1932} C_DIS
LIN {X 91.4696,Y -100.2039,Z 170,A -45.379,B 9.6538,C 0.3033,E1 9.7678,E2 496.4866} C_DIS
LIN {X 94.3303,Y -97.5148,Z 170,A -43.6978,B 9.6538,C 0.2993,E1 9.7712,E2 494.8009} C_DIS
LIN {X 97.4218,Y -94.4264,Z 170,A -41.8847,B 9.654,C 0.2961,E1 9.7747,E2 492.9899} C_DIS
LIN {X 100.3598,Y -91.2978,Z 170,A -40.1329,B 9.654,C 0.2935,E1 9.778,E2 491.2439} C_DIS
LIN {X 103.0897,Y -88.2045,Z 170,A -38.2963,B 9.6542,C 0.2873,E1 9.7814,E2 489.3936} C_DIS
LIN {X 106.1478,Y -84.4985,Z 170,A -36.3268,B 9.6543,C 0.284,E1 9.7849,E2 487.4295} C_DIS
LIN {X 108.899,Y -80.922,Z 170,A -34.4709,B 9.6544,C 0.2806,E1 9.788,E2 485.5778} C_DIS
LIN {X 111.6076,Y -77.1444,Z 170,A -32.5411,B 9.6546,C 0.2766,E1 9.7911,E2 483.6502} C_DIS
LIN {X 114.0326,Y -73.5126,Z 170,A -30.7097,B 9.6546,C 0.2723,E1 9.7939,E2 481.8184} C_DIS
LIN {X 116.3693,Y -69.7542,Z 170,A -28.7071,B 9.6549,C 0.2643,E1 9.7968,E2 479.7969} C_DIS
LIN {X 118.8315,Y -65.4714,Z 170,A -26.8066,B 9.6549,C 0.2634,E1 9.7994,E2 477.9177} C_DIS
LIN {X 120.7591,Y -61.8396,Z 170,A -25.2529,B 9.6549,C 0.2631,E1 9.8014,E2 476.3851} C_DIS
LIN {X 122.2864,Y -58.7617,Z 170,A -23.3961,B 9.6553,C 0.2495,E1 9.8037,E2 474.4754} C_DIS
LIN {X 123.8344,Y -55.4242,Z 170,A -22.3554,B 9.6551,C 0.2577,E1 9.8048,E2 473.4979} C_DIS
LIN {X 124.9527,Y -52.8585,Z 170,A -21.0013,B 9.6553,C 0.2503,E1 9.8063,E2 472.1208} C_DIS
LIN {X 126.3761,Y -49.3554,Z 170,A -19.4502,B 9.6553,C 0.247,E1 9.8079,E2 470.5738} C_DIS
LIN {X 127.7437,Y -45.6999,Z 170,A -17.8417,B 9.6554,C 0.2434,E1 9.8095,E2 468.9686} C_DIS
LIN {X 129.1393,Y -41.5932,Z 170,A -16.1765,B 9.6554,C 0.2423,E1 9.8109,E2 467.3224} C_DIS
LIN {X 130.2117,Y -38.1021,Z 170,A -14.5625,B 9.6556,C 0.2362,E1 9.8122,E2 465.6977} C_DIS
LIN {X 131.6248,Y -32.8941,Z 170,A -12.1641,B 9.6558,C 0.2269,E1 9.8139,E2 463.2819} C_DIS
LIN {X 132.5556,Y -28.913,Z 170,A -10.6041,B 9.6558,C 0.226,E1 9.8149,E2 461.7411} C_DIS
LIN {X 133.1848,Y -25.8622,Z 170,A -9.4723,B 9.6558,C 0.2266,E1 9.8155,E2 460.6309} C_DIS
LIN {X 133.7788,Y -22.5873,Z 170,A -7.9146,B 9.656,C 0.2189,E1 9.8163,E2 459.0527} C_DIS
LIN {X 134.3198,Y -19.1074,Z 170,A -6.4161,B 9.6561,C 0.2143,E1 9.8169,E2 457.5512} C_DIS
LIN {X 134.8629,Y -14.7983,Z 170,A -4.6682,B 9.6561,C 0.2111,E1 9.8175,E2 455.8123} C_DIS
LIN {X 135.1439,Y -11.9735,Z 170,A -3.4852,B 9.6563,C 0.2079,E1 9.8178,E2 454.6301} C_DIS
LIN {X 135.3921,Y -8.7216,Z 170,A -2.2846,B 9.6563,C 0.2082,E1 9.818,E2 453.4503} C_DIS
LIN {X 135.5682,Y -5.3124,Z 170,A -0.6082,B 9.6565,C 0.1983,E1 9.8182,E2 451.7431} C_DIS
LIN {X 135.6703,Y -0.8902,Z 170,A 1.0965,B 9.6565,C 0.1968,E1 9.8182,E2 450.057} C_DIS
LIN {X 135.6496,Y 2.4895,Z 170,A 2.6588,B 9.6566,C 0.1894,E1 9.8182,E2 448.4764} C_DIS
LIN {X 135.5335,Y 6.1667,Z 170,A 4.1898,B 9.6567,C 0.1854,E1 9.8181,E2 446.9468} C_DIS
LIN {X 135.2543,Y 10.667,Z 170,A 6.0903,B 9.6568,C 0.18,E1 9.8177,E2 445.0451} C_DIS
LIN {X 134.9171,Y 14.2953,Z 170,A 7.4025,B 9.6568,C 0.181,E1 9.8173,E2 443.7597} C_DIS
LIN {X 134.5917,Y 17.0959,Z 170,A 8.6112,B 9.6568,C 0.1771,E1 9.8169,E2 442.5477} C_DIS
LIN {X 134.2101,Y 19.8752,Z 170,A 9.9505,B 9.657,C 0.17,E1 9.8164,E2 441.1881} C_DIS
LIN {X 133.6083,Y 23.5758,Z 170,A 11.3802,B 9.657,C 0.1691,E1 9.8157,E2 439.7761} C_DIS
LIN {X 132.9683,Y 26.9506,Z 170,A 12.7867,B 9.657,C 0.1661,E1 9.8149,E2 438.3739} C_DIS
LIN {X 132.3604,Y 29.7957,Z 170,A 14.0526,B 9.6571,C 0.1617,E1 9.8142,E2 437.1023} C_DIS
LIN {X 131.5244,Y 33.2896,Z 170,A 15.5191,B 9.6571,C 0.1586,E1 9.8132,E2 435.6409} C_DIS
LIN {X 130.6299,Y 36.6427,Z 170,A 17.2185,B 9.6573,C 0.149,E1 9.8119,E2 433.9111} C_DIS
LIN {X 129.4187,Y 40.7184,Z 170,A 18.8453,B 9.6573,C 0.148,E1 9.8106,E2 432.3041} C_DIS
LIN {X 128.2232,Y 44.3358,Z 170,A 20.2771,B 9.6573,C 0.1478,E1 9.8093,E2 430.8931} C_DIS
LIN {X 127.3283,Y 46.8504,Z 170,A 21.3975,B 9.6574,C 0.1449,E1 9.8083,E2 429.7727} C_DIS
LIN {X 125.9843,Y 50.3481,Z 170,A 22.9766,B 9.6574,C 0.1407,E1 9.8067,E2 428.1928} C_DIS
LIN {X 124.8252,Y 53.1605,Z 170,A 24.3408,B 9.6575,C 0.1355,E1 9.8052,E2 426.8178} C_DIS
LIN {X 123.3106,Y 56.5814,Z 170,A 25.8345,B 9.6575,C 0.1333,E1 9.8035,E2 425.3337} C_DIS
LIN {X 121.7757,Y 59.8124,Z 170,A 27.3985,B 9.6576,C 0.1281,E1 9.8015,E2 423.762} C_DIS
LIN {X 119.4955,Y 64.2509,Z 170,A 29.9069,B 9.6578,C 0.1133,E1 9.7982,E2 421.2025} C_DIS
LIN {X 117.2583,Y 68.2487,Z 170,A 31.1364,B 9.6577,C 0.1251,E1 9.7966,E2 420.0594} C_DIS
LIN {X 115.6913,Y 70.8723,Z 170,A 32.641,B 9.6577,C 0.1169,E1 9.7944,E2 418.5277} C_DIS
LIN {X 113.3122,Y 74.617,Z 170,A 34.4252,B 9.6578,C 0.1144,E1 9.7917,E2 416.7535} C_DIS
LIN {X 111.1518,Y 77.7996,Z 170,A 36.1273,B 9.6578,C 0.1088,E1 9.789,E2 415.0409} C_DIS
LIN {X 108.5062,Y 81.4486,Z 170,A 38.0126,B 9.6579,C 0.1048,E1 9.7859,E2 413.1569} C_DIS
LIN {X 105.2119,Y 85.6613,Z 170,A 40.2092,B 9.6579,C 0.1011,E1 9.782,E2 410.9669} C_DIS
LIN {X 102.3948,Y 89.0096,Z 170,A 42.0672,B 9.658,C 0.0969,E1 9.7787,E2 409.1068} C_DIS
LIN {X 99.4291,Y 92.3105,Z 170,A 43.8556,B 9.658,C 0.0949,E1 9.7753,E2 407.3283} C_DIS
LIN {X 97.2002,Y 94.6553,Z 170,A 45.2799,B 9.658,C 0.0907,E1 9.7725,E2 405.8963} C_DIS
LIN {X 94.0017,Y 97.8323,Z 170,A 47.0995,B 9.658,C 0.0888,E1 9.7689,E2 404.0864} C_DIS
LIN {X 90.9431,Y 100.6817,Z 170,A 48.883,B 9.6581,C 0.085,E1 9.7652,E2 402.3002} C_DIS
LIN {X 87.5573,Y 103.64,Z 170,A 50.779,B 9.6581,C 0.0815,E1 9.7612,E2 400.404} C_DIS
LIN {X 84.3742,Y 106.2467,Z 170,A 52.4636,B 9.6581,C 0.0796,E1 9.7576,E2 398.7254} C_DIS
LIN {X 80.754,Y 109.0241,Z 170,A 54.3992,B 9.6581,C 0.0761,E1 9.7533,E2 396.7883} C_DIS
LIN {X 77.5066,Y 111.3556,Z 170,A 56.1857,B 9.6582,C 0.0711,E1 9.7492,E2 394.9895} C_DIS
LIN {X 73.2406,Y 114.2067,Z 170,A 58.1864,B 9.6582,C 0.0714,E1 9.7445,E2 393.009} C_DIS
LIN {X 70.7741,Y 115.7515,Z 170,A 59.7123,B 9.6582,C 0.063,E1 9.7408,E2 391.4464} C_DIS
LIN {X 67.5704,Y 117.651,Z 170,A 60.9864,B 9.6582,C 0.0674,E1 9.7378,E2 390.209} C_DIS
LIN {X 63.7978,Y 119.7385,Z 170,A 62.8125,B 9.6582,C 0.0648,E1 9.7333,E2 388.3821} C_DIS
LIN {X 60.634,Y 121.3704,Z 170,A 64.1404,B 9.6582,C 0.0667,E1 9.7301,E2 387.0756} C_DIS
LIN {X 57.4999,Y 122.8859,Z 170,A 65.7595,B 9.6582,C 0.0617,E1 9.7259,E2 385.4383} C_DIS
LIN {X 54.0935,Y 124.4218,Z 170,A 67.2536,B 9.6582,C 0.0617,E1 9.7221,E2 383.9545} C_DIS
LIN {X 49.9144,Y 126.1585,Z 170,A 69.1785,B 9.6583,C 0.0594,E1 9.7172,E2 382.0281} C_DIS
LIN {X 46.4412,Y 127.4765,Z 170,A 70.544,B 9.6583,C 0.0622,E1 9.7137,E2 380.6875} C_DIS
LIN {X 43.172,Y 128.6201,Z 170,A 72.1735,B 9.6583,C 0.0573,E1 9.7093,E2 379.0378} C_DIS
LIN {X 40.1782,Y 129.587,Z 170,A 73.6735,B 9.6583,C 0.0525,E1 9.7053,E2 377.5171} C_DIS
LIN {X 35.9773,Y 130.816,Z 170,A 75.4271,B 9.6583,C 0.0531,E1 9.7006,E2 375.7755} C_DIS
LIN {X 31.9256,Y 131.8622,Z 170,A 77.0137,B 9.6583,C 0.0558,E1 9.6963,E2 374.2112} C_DIS
LIN {X 29.2484,Y 132.4832,Z 170,A 78.3302,B 9.6583,C 0.0518,E1 9.6927,E2 372.8761} C_DIS
LIN {X 25.5154,Y 133.2511,Z 170,A 79.8281,B 9.6583,C 0.0532,E1 9.6886,E2 371.3921} C_DIS
LIN {X 22.2458,Y 133.8358,Z 170,A 81.2515,B 9.6583,C 0.0522,E1 9.6847,E2 369.9667} C_DIS
LIN {X 18.075,Y 134.4634,Z 170,A 83.05,B 9.6583,C 0.0511,E1 9.6797,E2 368.1666} C_DIS
LIN {X 14.7833,Y 134.8646,Z 170,A 84.2367,B 9.6583,C 0.0551,E1 9.6765,E2 367.0064} C_DIS
LIN {X 11.562,Y 135.1787,Z 170,A 85.8018,B 9.6583,C 0.0507,E1 9.6721,E2 365.4177} C_DIS
LIN {X 7.6091,Y 135.4606,Z 170,A 87.5102,B 9.6583,C 0.0497,E1 9.6673,E2 363.7058} C_DIS
LIN {X 3.7459,Y 135.6205,Z 170,A 89.082,B 9.6583,C 0.0509,E1 9.663,E2 362.142} C_DIS
LIN {X -0.3234,Y 135.6726,Z 170,A 90.655,B 9.6583,C 0.0539,E1 9.6586,E2 360.5876} C_DIS
LIN {X -3.6683,Y 135.6227,Z 170,A 92.2257,B 9.6583,C 0.0508,E1 9.6542,E2 358.9983} C_DIS
LIN {X -7.4136,Y 135.4708,Z 170,A 93.9553,B 9.6583,C 0.0481,E1 9.6493,E2 357.2517} C_DIS
LIN {X -11.45,Y 135.1881,Z 170,A 95.4514,B 9.6583,C 0.0528,E1 9.6452,E2 355.7823} C_DIS
LIN {X -13.9754,Y 134.9515,Z 170,A 96.4899,B 9.6583,C 0.0538,E1 9.6423,E2 354.7484} C_DIS
LIN {X -17.5331,Y 134.5344,Z 170,A 98.1011,B 9.6583,C 0.0524,E1 9.6378,E2 353.1261} C_DIS
LIN {X -21.1546,Y 134.0132,Z 170,A 99.6851,B 9.6583,C 0.0524,E1 9.6335,E2 351.5383} C_DIS
LIN {X -25.3718,Y 133.2786,Z 170,A 101.4645,B 9.6583,C 0.0539,E1 9.6286,E2 349.7634} C_DIS
LIN {X -28.2078,Y 132.7079,Z 170,A 102.6423,B 9.6583,C 0.0556,E1 9.6254,E2 348.5918} C_DIS
LIN {X -31.5129,Y 131.9617,Z 170,A 104.1316,B 9.6583,C 0.0554,E1 9.6213,E2 347.0964} C_DIS
LIN {X -34.2297,Y 131.285,Z 170,A 105.6625,B 9.6583,C 0.0495,E1 9.6171,E2 345.5239} C_DIS
LIN {X -37.5984,Y 130.3592,Z 170,A 106.9062,B 9.6583,C 0.0552,E1 9.6138,E2 344.3094} C_DIS
LIN {X -41.1474,Y 129.2817,Z 170,A 108.3576,B 9.6583,C 0.0589,E1 9.61,E2 342.8731} C_DIS
LIN {X -44.9527,Y 128.0093,Z 170,A 109.9885,B 9.6583,C 0.0618,E1 9.6057,E2 341.2513} C_DIS
LIN {X -49.534,Y 126.3066,Z 170,A 112.2745,B 9.6583,C 0.0597,E1 9.5997,E2 338.9399} C_DIS
LIN {X -53.4573,Y 124.6969,Z 170,A 113.9939,B 9.6583,C 0.0631,E1 9.5952,E2 337.2306} C_DIS
LIN {X -56.7182,Y 123.2473,Z 170,A 115.3545,B 9.6583,C 0.0678,E1 9.5918,E2 335.889} C_DIS
LIN {X -64.8205,Y 119.1876,Z 170,A 119.0602,B 9.6582,C 0.0753,E1 9.5827,E2 332.2016} C_DIS
LIN {X -68.166,Y 117.3064,Z 170,A 121.0699,B 9.6582,C 0.0704,E1 9.5777,E2 330.1462} C_DIS
LIN {X -71.8552,Y 115.0835,Z 170,A 122.9024,B 9.6582,C 0.0729,E1 9.5733,E2 328.3137} C_DIS
LIN {X -75.6669,Y 112.6145,Z 170,A 124.6938,B 9.6582,C 0.0784,E1 9.5692,E2 326.5395} C_DIS
LIN {X -78.0045,Y 111.0077,Z 170,A 126.0146,B 9.6582,C 0.0782,E1 9.5661,E2 325.2048} C_DIS
LIN {X -80.7397,Y 109.0347,Z 170,A 127.593,B 9.6582,C 0.0778,E1 9.5625,E2 323.609} C_DIS
LIN {X -84.6898,Y 105.9955,Z 170,A 129.5732,B 9.6582,C 0.084,E1 9.5582,E2 321.646} C_DIS
LIN {X -88.1123,Y 103.1681,Z 170,A 132.0545,B 9.6582,C 0.0763,E1 9.5528,E2 319.0923} C_DIS
LIN {X -92.0032,Y 99.7137,Z 170,A 133.8278,B 9.6581,C 0.0886,E1 9.5492,E2 317.3732} C_DIS
LIN {X -95.6726,Y 96.1982,Z 170,A 135.8658,B 9.6581,C 0.095,E1 9.5452,E2 315.3505} C_DIS
LIN {X -97.8741,Y 93.9579,Z 170,A 137.753,B 9.6581,C 0.0875,E1 9.5414,E2 313.3961} C_DIS
LIN {X -101.2915,Y 90.2634,Z 170,A 139.1075,B 9.6579,C 0.1063,E1 9.5391,E2 312.138} C_DIS
LIN {X -103.5381,Y 87.6771,Z 170,A 140.8643,B 9.6579,C 0.1039,E1 9.5358,E2 310.3449} C_DIS
LIN {X -106.4614,Y 84.1039,Z 170,A 142.8032,B 9.6579,C 0.1086,E1 9.5324,E2 308.4094} C_DIS
LIN {X -109.1236,Y 80.6196,Z 170,A 144.4865,B 9.6578,C 0.116,E1 9.5296,E2 306.7486} C_DIS
LIN {X -111.6101,Y 77.1408,Z 170,A 146.4754,B 9.6578,C 0.117,E1 9.5264,E2 304.7393} C_DIS
LIN {X -114.0029,Y 73.5583,Z 170,A 148.2866,B 9.6578,C 0.1217,E1 9.5236,E2 302.931} C_DIS
LIN {X -116.2431,Y 69.964,Z 170,A 150.1139,B 9.6577,C 0.1254,E1 9.5209,E2 301.1009} C_DIS
LIN {X -118.1908,Y 66.6206,Z 170,A 152.0595,B 9.6577,C 0.1241,E1 9.5182,E2 299.1189} C_DIS
LIN {X -119.8221,Y 63.6385,Z 170,A 153.2371,B 9.6576,C 0.1324,E1 9.5167,E2 297.9743} C_DIS
LIN {X -121.4898,Y 60.3921,Z 170,A 154.5927,B 9.6575,C 0.1397,E1 9.515,E2 296.643} C_DIS
LIN {X -122.6742,Y 57.9499,Z 170,A 156.0382,B 9.6575,C 0.1375,E1 9.5132,E2 295.1622} C_DIS
LIN {X -124.3361,Y 54.2917,Z 170,A 157.6691,B 9.6575,C 0.1432,E1 9.5114,E2 293.5411} C_DIS
LIN {X -125.7053,Y 51.0404,Z 170,A 158.9458,B 9.6573,C 0.151,E1 9.5101,E2 292.2921} C_DIS
LIN {X -127.2501,Y 47.0586,Z 170,A 161.2646,B 9.6573,C 0.1468,E1 9.5077,E2 289.9122} C_DIS
LIN {X -128.3306,Y 44.0259,Z 170,A 162.463,B 9.6573,C 0.1535,E1 9.5066,E2 288.7351} C_DIS
LIN {X -129.6656,Y 39.9215,Z 170,A 164.1817,B 9.6572,C 0.1604,E1 9.5052,E2 287.031} C_DIS
LIN {X -130.6233,Y 36.6666,Z 170,A 165.604,B 9.6571,C 0.1646,E1 9.5041,E2 285.6115} C_DIS
LIN {X -131.3545,Y 33.9591,Z 170,A 166.763,B 9.6571,C 0.1684,E1 9.5033,E2 284.4569} C_DIS
LIN {X -132.238,Y 30.3315,Z 170,A 168.5042,B 9.6571,C 0.17,E1 9.5021,E2 282.6972} C_DIS
LIN {X -133.0506,Y 26.5458,Z 170,A 170.2602,B 9.657,C 0.1726,E1 9.5011,E2 280.928} C_DIS
LIN {X -133.694,Y 23.0959,Z 170,A 171.6356,B 9.6568,C 0.1787,E1 9.5005,E2 279.5674} C_DIS
LIN {X -134.2022,Y 19.9308,Z 170,A 173.1325,B 9.6568,C 0.1801,E1 9.4998,E2 278.0542} C_DIS
LIN {X -134.7203,Y 16.0422,Z 170,A 174.5881,B 9.6567,C 0.1884,E1 9.4993,E2 276.6249} C_DIS
LIN {X -135.1779,Y 11.5705,Z 170,A 176.6588,B 9.6567,C 0.1909,E1 9.4988,E2 274.535} C_DIS
LIN {X -135.4744,Y 7.3429,Z 170,A 178.5253,B 9.6565,C 0.1948,E1 9.4985,E2 272.6609} C_DIS
LIN {X -135.6319,Y 3.3351,Z 170,A -179.7719,B 9.6565,C 0.1996,E1 9.4983,E2 270.9585} C_DIS
LIN {X -135.6706,Y -0.8456,Z 170,A -178.0175,B 9.6563,C 0.2049,E1 9.4983,E2 269.2073} C_DIS
LIN {X -135.583,Y -4.9321,Z 170,A -176.2634,B 9.6563,C 0.2095,E1 9.4984,E2 267.4514} C_DIS
LIN {X -135.4049,Y -8.5132,Z 170,A -174.7083,B 9.6562,C 0.2131,E1 9.4987,E2 265.8927} C_DIS
LIN {X -135.0633,Y -12.8397,Z 170,A -172.8082,B 9.6561,C 0.2172,E1 9.4992,E2 263.986} C_DIS
LIN {X -134.5606,Y -17.3336,Z 170,A -170.9484,B 9.6559,C 0.2236,E1 9.4998,E2 262.134} C_DIS
LIN {X -133.9831,Y -21.3494,Z 170,A -169.0669,B 9.6559,C 0.2256,E1 9.5006,E2 260.2333} C_DIS
LIN {X -133.3702,Y -24.8924,Z 170,A -167.5488,B 9.6558,C 0.2299,E1 9.5013,E2 258.7165} C_DIS
LIN {X -132.6035,Y -28.6915,Z 170,A -166.0494,B 9.6556,C 0.237,E1 9.5022,E2 257.2355} C_DIS
LIN {X -131.9205,Y -31.6836,Z 170,A -164.5834,B 9.6556,C 0.2376,E1 9.5031,E2 255.7495} C_DIS
LIN {X -129.8903,Y -39.1873,Z 170,A -161.1146,B 9.6554,C 0.2434,E1 9.5058,E2 252.2604} C_DIS
LIN {X -128.1153,Y -44.6469,Z 170,A -158.8563,B 9.6552,C 0.253,E1 9.5078,E2 250.0246} C_DIS
LIN {X -126.5731,Y -48.8485,Z 170,A -157.0909,B 9.655,C 0.2604,E1 9.5095,E2 248.2761} C_DIS
LIN {X -125.2973,Y -52.0335,Z 170,A -155.5329,B 9.655,C 0.2623,E1 9.5111,E2 246.7056} C_DIS
LIN {X -124.0296,Y -54.9879,Z 170,A -154.3034,B 9.6548,C 0.2681,E1 9.5125,E2 245.493} C_DIS
LIN {X -122.5838,Y -58.1391,Z 170,A -152.6024,B 9.6548,C 0.2677,E1 9.5145,E2 243.7636} C_DIS
LIN {X -120.9802,Y -61.4053,Z 170,A -151.0429,B 9.6548,C 0.2712,E1 9.5165,E2 242.2022} C_DIS
LIN {X -118.7914,Y -65.5439,Z 170,A -149.0046,B 9.6546,C 0.2751,E1 9.5192,E2 240.1576} C_DIS
LIN {X -116.6529,Y -69.2784,Z 170,A -147.1471,B 9.6545,C 0.2788,E1 9.5218,E2 238.2962} C_DIS
LIN {X -113.9722,Y -73.6057,Z 170,A -144.3836,B 9.6547,C 0.2727,E1 9.5261,E2 235.4569} C_DIS
LIN {X -110.9727,Y -78.054,Z 170,A -142.8531,B 9.6541,C 0.2916,E1 9.5284,E2 234.0199} C_DIS
LIN {X -108.2084,Y -81.8432,Z 170,A -140.7067,B 9.6541,C 0.293,E1 9.532,E2 231.8538} C_DIS
LIN {X -105.5774,Y -85.2101,Z 170,A -138.8697,B 9.654,C 0.2964,E1 9.5352,E2 230.0136} C_DIS
LIN {X -102.8702,Y -88.4595,Z 170,A -137.0645,B 9.6539,C 0.2999,E1 9.5384,E2 228.2068} C_DIS
LIN {X -100.1168,Y -91.5647,Z 170,A -135.293,B 9.6538,C 0.3032,E1 9.5417,E2 226.4337} C_DIS
LIN {X -97.167,Y -94.6895,Z 170,A -133.4331,B 9.6537,C 0.306,E1 9.5453,E2 224.5688} C_DIS
LIN {X -93.979,Y -97.854,Z 170,A -131.5073,B 9.6536,C 0.3092,E1 9.5492,E2 222.64} C_DIS
LIN {X -90.6423,Y -100.9522,Z 170,A -129.5769,B 9.6535,C 0.3127,E1 9.5532,E2 220.7093} C_DIS
LIN {X -87.2136,Y -103.9285,Z 170,A -127.544,B 9.6535,C 0.3139,E1 9.5575,E2 218.6624} C_DIS
LIN {X -83.2924,Y -107.097,Z 170,A -125.4941,B 9.6533,C 0.3191,E1 9.562,E2 216.6229} C_DIS
LIN {X -78.8078,Y -110.4386,Z 170,A -123.1431,B 9.6531,C 0.3231,E1 9.5673,E2 214.2737} C_DIS
LIN {X -75.3051,Y -112.8561,Z 170,A -121.3418,B 9.6531,C 0.3258,E1 9.5715,E2 212.4722} C_DIS
LIN {X -71.2611,Y -115.4526,Z 170,A -119.2486,B 9.653,C 0.3275,E1 9.5764,E2 210.3713} C_DIS
LIN {X -67.6101,Y -117.6282,Z 170,A -117.435,B 9.653,C 0.3296,E1 9.5808,E2 208.5555} C_DIS
LIN {X -64.0655,Y -119.5951,Z 170,A -115.8198,B 9.6528,C 0.3337,E1 9.5847,E2 206.9526} C_DIS
LIN {X -61.6758,Y -120.8425,Z 170,A -114.6035,B 9.6528,C 0.3336,E1 9.5878,E2 205.7264} C_DIS
LIN {X -57.6594,Y -122.8122,Z 170,A -112.6874,B 9.6528,C 0.3352,E1 9.5926,E2 203.8069} C_DIS
LIN {X -54.2917,Y -124.3361,Z 170,A -111.2361,B 9.6526,C 0.3391,E1 9.5963,E2 202.3693} C_DIS
LIN {X -51.0106,Y -125.7173,Z 170,A -109.7624,B 9.6526,C 0.3412,E1 9.6001,E2 200.8993} C_DIS
LIN {X -48.4343,Y -126.7341,Z 170,A -108.3947,B 9.6526,C 0.3383,E1 9.6037,E2 199.5066} C_DIS
LIN {X -44.7716,Y -128.0721,Z 170,A -106.9111,B 9.6524,C 0.343,E1 9.6075,E2 198.0433} C_DIS
LIN {X -40.5902,Y -129.4597,Z 170,A -104.853,B 9.6525,C 0.3405,E1 9.6131,E2 195.9601} C_DIS
LIN {X -36.3527,Y -130.711,Z 170,A -103.1273,B 9.6524,C 0.3446,E1 9.6177,E2 194.2517} C_DIS
LIN {X -32.6317,Y -131.6914,Z 170,A -101.4904,B 9.6524,C 0.3454,E1 9.6221,E2 192.613} C_DIS
LIN {X -29.4519,Y -132.4389,Z 170,A -100.018,B 9.6524,C 0.3442,E1 9.6261,E2 191.1285} C_DIS
LIN {X -25.7141,Y -133.2131,Z 170,A -98.504,B 9.6524,C 0.3469,E1 9.6303,E2 189.6264} C_DIS
LIN {X -22.4944,Y -133.7944,Z 170,A -97.2214,B 9.6522,C 0.3495,E1 9.6338,E2 188.3559} C_DIS
LIN {X -19.361,Y -134.2836,Z 170,A -95.8352,B 9.6522,C 0.3489,E1 9.6376,E2 186.9633} C_DIS
LIN {X -16.6923,Y -134.6428,Z 170,A -94.7185,B 9.6522,C 0.3496,E1 9.6407,E2 185.8489} C_DIS
LIN {X -13.0183,Y -135.0461,Z 170,A -93.0573,B 9.6522,C 0.3478,E1 9.6453,E2 184.1744} C_DIS
LIN {X -10.1966,Y -135.2888,Z 170,A -91.3997,B 9.6526,C 0.3382,E1 9.6501,E2 182.4577} C_DIS
LIN {X -5.9012,Y -135.5452,Z 170,A -89.5037,B 9.6526,C 0.3365,E1 9.6554,E2 180.551} C_DIS
LIN {X -1.2774,Y -135.6671,Z 170,A -87.8992,B 9.6524,C 0.3438,E1 9.6598,E2 178.99} C_DIS
LIN {X -1.2774,Y -135.6671,Z 170,A -87.8992,B 9.6524,C 0.3438,E1 9.6598,E2 178.99} C_DIS
Enddeposition()
LIN {X 0.9829,Y -136.5807,Z 170,A -87.5031,B 9.5862,C 0.3632,E1 9.5951,E2 178.7175} C_DIS
Startdeposition()
$VEL.CP = VEL_PRINT
LIN {X -1.5125,Y -136.5778,Z 170,A -88.7478,B 9.586,C 0.3674,E1 9.5915,E2 179.9879} C_DIS
LIN {X -4.4087,Y -136.5142,Z 170,A -89.9701,B 9.586,C 0.3676,E1 9.5881,E2 181.2116} C_DIS
LIN {X -7.477,Y -136.3806,Z 170,A -91.2565,B 9.586,C 0.3676,E1 9.5845,E2 182.4983} C_DIS
LIN {X -10.2874,Y -136.1964,Z 170,A -92.476,B 9.586,C 0.3683,E1 9.5811,E2 183.723} C_DIS
LIN {X -13.8316,Y -135.884,Z 170,A -93.9367,B 9.586,C 0.3674,E1 9.577,E2 185.1803} C_DIS
LIN {X -16.9626,Y -135.5288,Z 170,A -95.2629,B 9.586,C 0.3672,E1 9.5733,E2 186.5076} C_DIS
LIN {X -19.6214,Y -135.1674,Z 170,A -96.4359,B 9.586,C 0.3678,E1 9.5701,E2 187.6869} C_DIS
LIN {X -23.2694,Y -134.5894,Z 170,A -97.9464,B 9.586,C 0.3665,E1 9.5659,E2 189.193} C_DIS
LIN {X -26.1007,Y -134.0675,Z 170,A -99.1528,B 9.586,C 0.366,E1 9.5626,E2 190.3995} C_DIS
LIN {X -29.4642,Y -133.3694,Z 170,A -100.6065,B 9.586,C 0.3655,E1 9.5586,E2 191.8551} C_DIS
LIN {X -32.8032,Y -132.5886,Z 170,A -102.0509,B 9.586,C 0.3649,E1 9.5547,E2 193.3007} C_DIS
LIN {X -35.8292,Y -131.8021,Z 170,A -103.3515,B 9.5861,C 0.3638,E1 9.5512,E2 194.6002} C_DIS
LIN {X -39.1755,Y -130.8475,Z 170,A -104.8365,B 9.5861,C 0.3633,E1 9.5472,E2 196.0887} C_DIS
LIN {X -42.3577,Y -129.8522,Z 170,A -106.2423,B 9.5861,C 0.3624,E1 9.5435,E2 197.4956} C_DIS
LIN {X -45.3065,Y -128.8517,Z 170,A -107.555,B 9.5862,C 0.3614,E1 9.54,E2 198.8092} C_DIS
LIN {X -48.5446,Y -127.6673,Z 170,A -109.0117,B 9.5862,C 0.3603,E1 9.5362,E2 200.2674} C_DIS
LIN {X -51.851,Y -126.3616,Z 170,A -110.5123,B 9.5863,C 0.359,E1 9.5323,E2 201.7693} C_DIS
LIN {X -54.9869,Y -125.0288,Z 170,A -111.951,B 9.5863,C 0.3577,E1 9.5286,E2 203.2093} C_DIS
LIN {X -57.9517,Y -123.6815,Z 170,A -113.3267,B 9.5864,C 0.3564,E1 9.5251,E2 204.5862} C_DIS
LIN {X -61.0461,Y -122.1838,Z 170,A -114.8427,B 9.5864,C 0.3561,E1 9.5213,E2 206.1114} C_DIS
LIN {X -64.9512,Y -120.1543,Z 170,A -116.7286,B 9.5864,C 0.3546,E1 9.5166,E2 208.0023} C_DIS
LIN {X -68.8067,Y -117.9891,Z 170,A -118.6338,B 9.5865,C 0.3531,E1 9.512,E2 209.9136} C_DIS
LIN {X -72.5337,Y -115.7352,Z 170,A -120.4514,B 9.5866,C 0.3503,E1 9.5077,E2 211.7299} C_DIS
LIN {X -76.1292,Y -113.4021,Z 170,A -122.1653,B 9.5868,C 0.346,E1 9.5037,E2 213.4329} C_DIS
LIN {X -79.0155,Y -111.4103,Z 170,A -123.7002,B 9.5868,C 0.3449,E1 9.5002,E2 214.9756} C_DIS
LIN {X -82.5583,Y -108.811,Z 170,A -125.5116,B 9.587,C 0.3412,E1 9.4961,E2 216.7826} C_DIS
LIN {X -85.6313,Y -106.409,Z 170,A -127.2482,B 9.587,C 0.3403,E1 9.4923,E2 218.5314} C_DIS
LIN {X -88.6519,Y -103.9061,Z 170,A -128.8978,B 9.587,C 0.3375,E1 9.4888,E2 220.1811} C_DIS
LIN {X -92.0449,Y -100.9131,Z 170,A -130.8124,B 9.5872,C 0.3342,E1 9.4848,E2 222.0972} C_DIS
LIN {X -95.261,Y -97.8829,Z 170,A -132.6235,B 9.5874,C 0.3299,E1 9.4811,E2 223.9024} C_DIS
LIN {X -97.9418,Y -95.2001,Z 170,A -134.3366,B 9.5874,C 0.329,E1 9.4778,E2 225.6301} C_DIS
LIN {X -100.8552,Y -92.1086,Z 170,A -136.1375,B 9.5874,C 0.3256,E1 9.4743,E2 227.4327} C_DIS
LIN {X -103.7662,Y -88.8162,Z 170,A -137.9719,B 9.5876,C 0.3216,E1 9.471,E2 229.2652} C_DIS
LIN {X -106.5386,Y -85.4707,Z 170,A -139.7413,B 9.5878,C 0.3166,E1 9.4679,E2 231.0271} C_DIS
LIN {X -108.7594,Y -82.6267,Z 170,A -141.255,B 9.5879,C 0.3132,E1 9.4653,E2 232.5402} C_DIS
LIN {X -110.8129,Y -79.8513,Z 170,A -142.8183,B 9.5879,C 0.312,E1 9.4627,E2 234.117} C_DIS
LIN {X -113.3548,Y -76.2001,Z 170,A -144.6098,B 9.5881,C 0.3062,E1 9.4599,E2 235.8982} C_DIS
LIN {X -115.1693,Y -73.4281,Z 170,A -146.0864,B 9.5881,C 0.3045,E1 9.4576,E2 237.3848} C_DIS
LIN {X -117.5051,Y -69.6294,Z 170,A -147.9192,B 9.5883,C 0.2993,E1 9.455,E2 239.2119} C_DIS
LIN {X -119.2798,Y -66.544,Z 170,A -149.4526,B 9.5884,C 0.2963,E1 9.4529,E2 240.7494} C_DIS
LIN {X -121.2491,Y -62.8823,Z 170,A -151.1831,B 9.5886,C 0.2916,E1 9.4506,E2 242.477} C_DIS
LIN {X -122.6601,Y -60.0807,Z 170,A -152.5699,B 9.5886,C 0.2895,E1 9.4489,E2 243.8716} C_DIS
LIN {X -124.3307,Y -56.5477,Z 170,A -154.1917,B 9.5888,C 0.2849,E1 9.447,E2 245.4903} C_DIS
LIN {X -125.5,Y -53.8973,Z 170,A -155.4232,B 9.5888,C 0.282,E1 9.4456,E2 246.7228} C_DIS
LIN {X -126.9344,Y -50.4299,Z 170,A -157.0143,B 9.589,C 0.2781,E1 9.4439,E2 248.315} C_DIS
LIN {X -128.2019,Y -47.1173,Z 170,A -158.5256,B 9.589,C 0.2746,E1 9.4424,E2 249.8281} C_DIS
LIN {X -129.3232,Y -43.9464,Z 170,A -159.9559,B 9.5892,C 0.2711,E1 9.4411,E2 251.2598} C_DIS
LIN {X -130.3108,Y -40.9221,Z 170,A -161.308,B 9.5892,C 0.2677,E1 9.44,E2 252.6129} C_DIS
LIN {X -131.2684,Y -37.7379,Z 170,A -162.7276,B 9.5894,C 0.2643,E1 9.4389,E2 254.0344} C_DIS
LIN {X -132.1842,Y -34.3963,Z 170,A -164.1959,B 9.5894,C 0.2605,E1 9.4378,E2 255.5034} C_DIS
LIN {X -132.83,Y -31.8014,Z 170,A -165.3528,B 9.5895,C 0.2579,E1 9.437,E2 256.6637} C_DIS
LIN {X -133.5454,Y -28.649,Z 170,A -166.7362,B 9.5896,C 0.2546,E1 9.4362,E2 258.0493} C_DIS
LIN {X -134.3059,Y -24.8536,Z 170,A -168.354,B 9.5898,C 0.2499,E1 9.4353,E2 259.6652} C_DIS
LIN {X -134.8276,Y -21.8419,Z 170,A -169.6397,B 9.5898,C 0.2463,E1 9.4347,E2 260.9501} C_DIS
LIN {X -135.2507,Y -19.0384,Z 170,A -170.8772,B 9.5899,C 0.2437,E1 9.4342,E2 262.1924} C_DIS
LIN {X -135.6976,Y -15.5476,Z 170,A -172.3614,B 9.59,C 0.2396,E1 9.4337,E2 263.6763} C_DIS
LIN {X -135.9974,Y -12.6502,Z 170,A -173.5871,B 9.59,C 0.2361,E1 9.4334,E2 264.9013} C_DIS
LIN {X -136.2481,Y -9.5789,Z 170,A -174.9099,B 9.5902,C 0.2329,E1 9.4331,E2 266.2266} C_DIS
LIN {X -136.4266,Y -6.5625,Z 170,A -176.2218,B 9.5902,C 0.23,E1 9.4329,E2 267.5428} C_DIS
LIN {X -136.5525,Y -3.0317,Z 170,A -177.8431,B 9.5902,C 0.2281,E1 9.4328,E2 269.1798} C_DIS
LIN {X -136.5822,Y 0.8692,Z 170,A -179.3947,B 9.5904,C 0.2219,E1 9.4328,E2 270.7194} C_DIS
LIN {X -136.5284,Y 3.8989,Z 170,A 179.301,B 9.5905,C 0.2187,E1 9.4328,E2 272.0265} C_DIS
LIN {X -136.3806,Y 7.477,Z 170,A 177.8214,B 9.5906,C 0.214,E1 9.4331,E2 273.5019} C_DIS
LIN {X -136.1759,Y 10.5681,Z 170,A 176.4938,B 9.5906,C 0.2107,E1 9.4333,E2 274.8317} C_DIS
LIN {X -135.884,Y 13.8316,Z 170,A 175.1006,B 9.5908,C 0.207,E1 9.4337,E2 276.2258} C_DIS
LIN {X -135.5788,Y 16.543,Z 170,A 173.9116,B 9.5908,C 0.2045,E1 9.4341,E2 277.419} C_DIS
LIN {X -135.0977,Y 20.1093,Z 170,A 172.3997,B 9.5909,C 0.2002,E1 9.4347,E2 278.9298} C_DIS
LIN {X -134.5894,Y 23.2694,Z 170,A 171.0341,B 9.5909,C 0.1967,E1 9.4353,E2 280.2968} C_DIS
LIN {X -134.0321,Y 26.2857,Z 170,A 169.7193,B 9.591,C 0.1935,E1 9.436,E2 281.6137} C_DIS
LIN {X -133.3718,Y 29.4534,Z 170,A 168.3434,B 9.5911,C 0.1899,E1 9.4368,E2 282.9904} C_DIS
LIN {X -132.5886,Y 32.8032,Z 170,A 166.8767,B 9.5911,C 0.1862,E1 9.4378,E2 284.4585} C_DIS
LIN {X -131.8007,Y 35.8345,Z 170,A 165.5402,B 9.5912,C 0.1829,E1 9.4387,E2 285.7964} C_DIS
LIN {X -130.8475,Y 39.1755,Z 170,A 164.0584,B 9.5913,C 0.1792,E1 9.4399,E2 287.2797} C_DIS
LIN {X -129.963,Y 42.0109,Z 170,A 162.8025,B 9.5913,C 0.1759,E1 9.4409,E2 288.5353} C_DIS
LIN {X -128.8267,Y 45.3786,Z 170,A 161.2763,B 9.5914,C 0.1724,E1 9.4423,E2 290.0643} C_DIS
LIN {X -127.6673,Y 48.5446,Z 170,A 159.8393,B 9.5915,C 0.1689,E1 9.4437,E2 291.5026} C_DIS
LIN {X -126.563,Y 51.3513,Z 170,A 158.5245,B 9.5915,C 0.1663,E1 9.4451,E2 292.8221} C_DIS
LIN {X -125.0288,Y 54.9869,Z 170,A 156.8727,B 9.5916,C 0.1618,E1 9.4469,E2 294.4717} C_DIS
LIN {X -123.6815,Y 57.9517,Z 170,A 155.4854,B 9.5916,C 0.1585,E1 9.4485,E2 295.8602} C_DIS
LIN {X -122.1838,Y 61.0461,Z 170,A 154.0358,B 9.5917,C 0.1548,E1 9.4503,E2 297.3091} C_DIS
LIN {X -120.5239,Y 64.2632,Z 170,A 152.4881,B 9.5917,C 0.1514,E1 9.4523,E2 298.8588} C_DIS
LIN {X -118.8961,Y 67.2267,Z 170,A 151.0315,B 9.5918,C 0.1484,E1 9.4543,E2 300.3186} C_DIS
LIN {X -117.1028,Y 70.3044,Z 170,A 149.5332,B 9.5918,C 0.1447,E1 9.4564,E2 301.8157} C_DIS
LIN {X -115.2692,Y 73.2721,Z 170,A 147.9708,B 9.5919,C 0.1428,E1 9.4588,E2 303.3887} C_DIS
LIN {X -112.8638,Y 76.9256,Z 170,A 146.0585,B 9.5919,C 0.1397,E1 9.4618,E2 305.3084} C_DIS
LIN {X -110.4554,Y 80.3445,Z 170,A 144.3763,B 9.592,C 0.1342,E1 9.4645,E2 306.9799} C_DIS
LIN {X -108.2768,Y 83.2577,Z 170,A 142.7526,B 9.592,C 0.1324,E1 9.4672,E2 308.6139} C_DIS
LIN {X -105.5354,Y 86.7063,Z 170,A 140.9751,B 9.5921,C 0.1269,E1 9.4703,E2 310.3809} C_DIS
LIN {X -102.9184,Y 89.7964,Z 170,A 139.2071,B 9.5921,C 0.1243,E1 9.4736,E2 312.1557} C_DIS
LIN {X -100.2573,Y 92.7591,Z 170,A 137.5741,B 9.5922,C 0.12,E1 9.4766,E2 313.7824} C_DIS
LIN {X -97.6411,Y 95.5082,Z 170,A 135.8693,B 9.5922,C 0.1186,E1 9.48,E2 315.4992} C_DIS
LIN {X -94.6877,Y 98.4378,Z 170,A 134.2075,B 9.5923,C 0.1135,E1 9.4833,E2 317.1492} C_DIS
LIN {X -92.1719,Y 100.797,Z 170,A 132.7276,B 9.5923,C 0.1112,E1 9.4863,E2 318.6317} C_DIS
LIN {X -89.5341,Y 103.1472,Z 170,A 131.1501,B 9.5923,C 0.1101,E1 9.4896,E2 320.2193} C_DIS
LIN {X -86.09,Y 106.0391,Z 170,A 129.3338,B 9.5924,C 0.1052,E1 9.4935,E2 322.0253} C_DIS
LIN {X -83.3936,Y 108.1722,Z 170,A 127.8686,B 9.5924,C 0.103,E1 9.4967,E2 323.4919} C_DIS
LIN {X -80.0734,Y 110.6519,Z 170,A 126.0763,B 9.5924,C 0.1009,E1 9.5008,E2 325.289} C_DIS
LIN {X -76.9926,Y 112.8178,Z 170,A 124.5217,B 9.5924,C 0.0978,E1 9.5043,E2 326.8393} C_DIS
LIN {X -74.0079,Y 114.7981,Z 170,A 123.0238,B 9.5925,C 0.0953,E1 9.5078,E2 328.3352} C_DIS
LIN {X -71.0498,Y 116.652,Z 170,A 121.548,B 9.5925,C 0.0932,E1 9.5113,E2 329.8111} C_DIS
LIN {X -68.1278,Y 118.3821,Z 170,A 120.0956,B 9.5925,C 0.0916,E1 9.5148,E2 331.2656} C_DIS
LIN {X -65.0004,Y 120.1279,Z 170,A 118.4614,B 9.5925,C 0.0919,E1 9.5189,E2 332.9144} C_DIS
LIN {X -61.346,Y 122.0335,Z 170,A 116.8462,B 9.5925,C 0.0874,E1 9.5229,E2 334.5144} C_DIS
LIN {X -58.1032,Y 123.6115,Z 170,A 115.3296,B 9.5925,C 0.0856,E1 9.5267,E2 336.0302} C_DIS
LIN {X -55.4012,Y 124.8436,Z 170,A 114.0526,B 9.5926,C 0.0846,E1 9.5299,E2 337.3099} C_DIS
LIN {X -52.0039,Y 126.2977,Z 170,A 112.5188,B 9.5926,C 0.0825,E1 9.5339,E2 338.8406} C_DIS
LIN {X -48.6986,Y 127.6096,Z 170,A 111.0198,B 9.5926,C 0.081,E1 9.5378,E2 340.3393} C_DIS
LIN {X -45.5331,Y 128.7731,Z 170,A 109.5991,B 9.5926,C 0.0797,E1 9.5415,E2 341.7597} C_DIS
LIN {X -42.916,Y 129.6663,Z 170,A 108.4387,B 9.5926,C 0.0786,E1 9.5446,E2 342.9192} C_DIS
LIN {X -39.6905,Y 130.6898,Z 170,A 106.9732,B 9.5926,C 0.0782,E1 9.5485,E2 344.3892} C_DIS
LIN {X -35.9896,Y 131.7593,Z 170,A 105.3892,B 9.5926,C 0.0763,E1 9.5527,E2 345.9683} C_DIS
LIN {X -33.3403,Y 132.4522,Z 170,A 104.2106,B 9.5926,C 0.076,E1 9.5559,E2 347.1496} C_DIS
LIN {X -29.6191,Y 133.336,Z 170,A 102.6297,B 9.5926,C 0.0744,E1 9.5602,E2 348.7267} C_DIS
LIN {X -26.5949,Y 133.9711,Z 170,A 101.3261,B 9.5926,C 0.0738,E1 9.5638,E2 350.0303} C_DIS
LIN {X -23.4237,Y 134.5618,Z 170,A 99.9762,B 9.5927,C 0.073,E1 9.5675,E2 351.379} C_DIS
LIN {X -20.7343,Y 135.0009,Z 170,A 98.8347,B 9.5927,C 0.0724,E1 9.5706,E2 352.5195} C_DIS
LIN {X -17.5524,Y 135.4515,Z 170,A 97.4353,B 9.5927,C 0.0728,E1 9.5745,E2 353.9244} C_DIS
LIN {X -13.8316,Y 135.884,Z 170,A 95.9118,B 9.5927,C 0.0713,E1 9.5787,E2 355.4413} C_DIS
LIN {X -10.8703,Y 136.1521,Z 170,A 94.6599,B 9.5927,C 0.0711,E1 9.5822,E2 356.6931} C_DIS
LIN {X -7.6268,Y 136.3731,Z 170,A 93.302,B 9.5927,C 0.0707,E1 9.586,E2 358.0496} C_DIS
LIN {X -5.0824,Y 136.4896,Z 170,A 92.1852,B 9.5927,C 0.0715,E1 9.5891,E2 359.1717} C_DIS
LIN {X -1.5125,Y 136.5778,Z 170,A 90.7392,B 9.5927,C 0.0703,E1 9.5932,E2 360.6107} C_DIS
LIN {X 1.5125,Y 136.5778,Z 170,A 89.4687,B 9.5927,C 0.0703,E1 9.5967,E2 361.8808} C_DIS
LIN {X 4.4087,Y 136.5142,Z 170,A 88.2464,B 9.5927,C 0.0705,E1 9.6001,E2 363.1034} C_DIS
LIN {X 7.477,Y 136.3806,Z 170,A 86.996,B 9.5927,C 0.0699,E1 9.6036,E2 364.3488} C_DIS
LIN {X 10.2216,Y 136.2012,Z 170,A 85.7606,B 9.5927,C 0.0718,E1 9.6071,E2 365.5936} C_DIS
LIN {X 13.8316,Y 135.884,Z 170,A 84.2855,B 9.5927,C 0.0712,E1 9.6111,E2 367.0627} C_DIS
LIN {X 16.507,Y 135.5831,Z 170,A 83.1169,B 9.5927,C 0.0724,E1 9.6144,E2 368.2355} C_DIS
LIN {X 20.1093,Y 135.0977,Z 170,A 81.6314,B 9.5927,C 0.0721,E1 9.6185,E2 369.7159} C_DIS
LIN {X 24.3895,Y 134.389,Z 170,A 79.7837,B 9.5927,C 0.0735,E1 9.6236,E2 371.5664} C_DIS
LIN {X 28.0288,Y 133.6793,Z 170,A 78.2595,B 9.5927,C 0.0738,E1 9.6277,E2 373.0864} C_DIS
LIN {X 31.0557,Y 133.0078,Z 170,A 76.9624,B 9.5927,C 0.0745,E1 9.6313,E2 374.3828} C_DIS
LIN {X 34.2342,Y 132.2254,Z 170,A 75.5906,B 9.5927,C 0.0754,E1 9.635,E2 375.7541} C_DIS
LIN {X 37.4277,Y 131.3572,Z 170,A 74.2009,B 9.5927,C 0.0765,E1 9.6387,E2 377.1438} C_DIS
LIN {X 40.596,Y 130.4127,Z 170,A 72.8401,B 9.5927,C 0.077,E1 9.6424,E2 378.5012} C_DIS
LIN {X 43.444,Y 129.4905,Z 170,A 71.5711,B 9.5927,C 0.0784,E1 9.6457,E2 379.7715} C_DIS
LIN {X 46.963,Y 128.2575,Z 170,A 70.0137,B 9.5927,C 0.0798,E1 9.6498,E2 381.328} C_DIS
LIN {X 50.123,Y 127.0559,Z 170,A 68.5961,B 9.5927,C 0.0812,E1 9.6535,E2 382.7454} C_DIS
LIN {X 53.4212,Y 125.7058,Z 170,A 67.1136,B 9.5927,C 0.0826,E1 9.6573,E2 384.2264} C_DIS
LIN {X 56.3451,Y 124.4214,Z 170,A 65.7939,B 9.5927,C 0.0837,E1 9.6607,E2 385.5436} C_DIS
LIN {X 59.5019,Y 122.9432,Z 170,A 64.3263,B 9.5926,C 0.0856,E1 9.6644,E2 387.0118} C_DIS
LIN {X 62.7333,Y 121.3273,Z 170,A 62.7722,B 9.5926,C 0.0884,E1 9.6683,E2 388.5706} C_DIS
LIN {X 66.4701,Y 119.3207,Z 170,A 60.9841,B 9.5926,C 0.091,E1 9.6727,E2 390.36} C_DIS
LIN {X 70.3044,Y 117.1028,Z 170,A 59.1224,B 9.5926,C 0.0937,E1 9.6771,E2 392.2223} C_DIS
LIN {X 74.0079,Y 114.7981,Z 170,A 57.3905,B 9.5926,C 0.0944,E1 9.6812,E2 393.9424} C_DIS
LIN {X 77.0976,Y 112.7457,Z 170,A 55.7444,B 9.5925,C 0.0989,E1 9.685,E2 395.5998} C_DIS
LIN {X 80.4416,Y 110.385,Z 170,A 54.1195,B 9.5925,C 0.0997,E1 9.6887,E2 397.2137} C_DIS
LIN {X 83.8229,Y 107.8394,Z 170,A 52.3294,B 9.5925,C 0.1031,E1 9.6927,E2 399.006} C_DIS
LIN {X 87.3082,Y 105.0377,Z 170,A 50.4594,B 9.5924,C 0.1063,E1 9.6967,E2 400.8757} C_DIS
LIN {X 90.7319,Y 102.0952,Z 170,A 48.6499,B 9.5924,C 0.108,E1 9.7005,E2 402.6755} C_DIS
LIN {X 93.4058,Y 99.655,Z 170,A 47.1554,B 9.5924,C 0.1104,E1 9.7036,E2 404.1676} C_DIS
LIN {X 96.1794,Y 96.98,Z 170,A 45.4573,B 9.5923,C 0.1155,E1 9.707,E2 405.8761} C_DIS
LIN {X 99.0485,Y 94.0487,Z 170,A 43.854,B 9.5923,C 0.1164,E1 9.7101,E2 407.4657} C_DIS
LIN {X 101.4489,Y 91.4543,Z 170,A 42.299,B 9.5923,C 0.1212,E1 9.713,E2 409.0302} C_DIS
LIN {X 104.3514,Y 88.1281,Z 170,A 40.5494,B 9.5922,C 0.1229,E1 9.7162,E2 410.768} C_DIS
LIN {X 106.5386,Y 85.4707,Z 170,A 39.0496,B 9.5922,C 0.1274,E1 9.7188,E2 412.2754} C_DIS
LIN {X 109.2058,Y 82.0351,Z 170,A 37.2331,B 9.5921,C 0.1314,E1 9.7219,E2 414.0917} C_DIS
LIN {X 111.8669,Y 78.3682,Z 170,A 35.445,B 9.5921,C 0.1333,E1 9.7248,E2 415.867} C_DIS
LIN {X 113.808,Y 75.5213,Z 170,A 33.9393,B 9.592,C 0.1381,E1 9.7272,E2 417.3809} C_DIS
LIN {X 116.1961,Y 71.793,Z 170,A 32.0865,B 9.592,C 0.1425,E1 9.7299,E2 419.2342} C_DIS
LIN {X 118.3821,Y 68.1278,Z 170,A 30.4118,B 9.592,C 0.1443,E1 9.7323,E2 420.8958} C_DIS
LIN {X 120.1543,Y 64.9512,Z 170,A 28.8039,B 9.5918,C 0.1501,E1 9.7344,E2 422.5146} C_DIS
LIN {X 121.9454,Y 61.519,Z 170,A 27.2926,B 9.5918,C 0.1516,E1 9.7363,E2 424.0131} C_DIS
LIN {X 123.4418,Y 58.4584,Z 170,A 25.9214,B 9.5918,C 0.1539,E1 9.738,E2 425.378} C_DIS
LIN {X 124.8385,Y 55.4125,Z 170,A 24.497,B 9.5917,C 0.1581,E1 9.7396,E2 426.8058} C_DIS
LIN {X 126.2977,Y 52.0039,Z 170,A 22.9989,B 9.5917,C 0.1609,E1 9.7413,E2 428.2979} C_DIS
LIN {X 127.6096,Y 48.6986,Z 170,A 21.5212,B 9.5916,C 0.1646,E1 9.7428,E2 429.7749} C_DIS
LIN {X 128.7731,Y 45.5331,Z 170,A 20.1285,B 9.5916,C 0.1679,E1 9.7441,E2 431.166} C_DIS
LIN {X 129.7146,Y 42.7709,Z 170,A 18.9014,B 9.5915,C 0.1713,E1 9.7452,E2 432.3944} C_DIS
LIN {X 130.8,Y 39.3305,Z 170,A 17.4343,B 9.5915,C 0.1744,E1 9.7464,E2 433.857} C_DIS
LIN {X 131.6197,Y 36.4889,Z 170,A 16.2273,B 9.5914,C 0.1771,E1 9.7473,E2 435.0607} C_DIS
LIN {X 132.4763,Y 33.2455,Z 170,A 14.8038,B 9.5913,C 0.1814,E1 9.7483,E2 436.4874} C_DIS
LIN {X 133.336,Y 29.6191,Z 170,A 13.2912,B 9.5913,C 0.1847,E1 9.7492,E2 437.9951} C_DIS
LIN {X 134.2061,Y 25.3758,Z 170,A 11.5128,B 9.5911,C 0.1889,E1 9.7502,E2 439.7701} C_DIS
LIN {X 134.8276,Y 21.8419,Z 170,A 10.0242,B 9.5911,C 0.1928,E1 9.7509,E2 441.258} C_DIS
LIN {X 135.3009,Y 18.6875,Z 170,A 8.7083,B 9.591,C 0.1961,E1 9.7514,E2 442.5724} C_DIS
LIN {X 135.6976,Y 15.5476,Z 170,A 7.3982,B 9.591,C 0.1995,E1 9.7519,E2 443.8815} C_DIS
LIN {X 136.0191,Y 12.4247,Z 170,A 6.128,B 9.5909,C 0.2022,E1 9.7522,E2 445.147} C_DIS
LIN {X 136.278,Y 9.1702,Z 170,A 4.7625,B 9.5908,C 0.2061,E1 9.7525,E2 446.5133} C_DIS
LIN {X 136.4504,Y 6.089,Z 170,A 3.4899,B 9.5908,C 0.2094,E1 9.7527,E2 447.7844} C_DIS
LIN {X 136.5525,Y 3.0317,Z 170,A 2.0843,B 9.5906,C 0.216,E1 9.7527,E2 449.2065} C_DIS
LIN {X 136.5822,Y -0.8692,Z 170,A 0.5259,B 9.5905,C 0.2189,E1 9.7527,E2 450.7567} C_DIS
LIN {X 136.5142,Y -4.4087,Z 170,A -0.8523,B 9.5905,C 0.2207,E1 9.7527,E2 452.123} C_DIS
LIN {X 136.3806,Y -7.477,Z 170,A -2.1187,B 9.5904,C 0.2239,E1 9.7525,E2 453.388} C_DIS
LIN {X 136.1759,Y -10.5681,Z 170,A -3.4057,B 9.5904,C 0.2274,E1 9.7522,E2 454.6748} C_DIS
LIN {X 135.884,Y -13.8316,Z 170,A -4.7564,B 9.5902,C 0.2309,E1 9.7519,E2 456.0238} C_DIS
LIN {X 135.5983,Y -16.3798,Z 170,A -5.8358,B 9.5902,C 0.2341,E1 9.7515,E2 457.1047} C_DIS
LIN {X 135.0977,Y -20.1093,Z 170,A -7.3749,B 9.5901,C 0.2377,E1 9.7509,E2 458.6406} C_DIS
LIN {X 134.5894,Y -23.2694,Z 170,A -8.6991,B 9.59,C 0.2412,E1 9.7503,E2 459.9638} C_DIS
LIN {X 134.0321,Y -26.2857,Z 170,A -9.9581,B 9.5899,C 0.2442,E1 9.7497,E2 461.2207} C_DIS
LIN {X 133.3694,Y -29.4642,Z 170,A -11.3126,B 9.5899,C 0.2479,E1 9.7489,E2 462.5756} C_DIS
LIN {X 132.5886,Y -32.8032,Z 170,A -12.7311,B 9.5897,C 0.2516,E1 9.748,E2 463.9932} C_DIS
LIN {X 131.8007,Y -35.8345,Z 170,A -14.0277,B 9.5897,C 0.2549,E1 9.747,E2 465.2891} C_DIS
LIN {X 130.8475,Y -39.1755,Z 170,A -15.4656,B 9.5895,C 0.2585,E1 9.7459,E2 466.726} C_DIS
LIN {X 129.9979,Y -41.9018,Z 170,A -16.6865,B 9.5895,C 0.2624,E1 9.7449,E2 467.951} C_DIS
Enddeposition()
END
